aff1Si[0  , 0] := 1.00000E+01; aff1Si[0  , 1] := -9.41486E+00;
aff1Si[1  , 0] := 1.99800E+01; aff1Si[1  , 1] := -1.02392E+01;
aff1Si[2  , 0] := 2.99600E+01; aff1Si[2  , 1] := -1.04800E+01;
aff1Si[3  , 0] := 3.99400E+01; aff1Si[3  , 1] := -1.06753E+01;
aff1Si[4  , 0] := 4.99200E+01; aff1Si[4  , 1] := -1.09200E+01;
aff1Si[5  , 0] := 5.99000E+01; aff1Si[5  , 1] := -1.12738E+01;
aff1Si[6  , 0] := 6.98800E+01; aff1Si[6  , 1] := -1.18088E+01;
aff1Si[7  , 0] := 7.98600E+01; aff1Si[7  , 1] := -1.26670E+01;
aff1Si[8  , 0] := 8.98400E+01; aff1Si[8  , 1] := -1.42966E+01;
aff1Si[9  , 0] := 9.98200E+01; aff1Si[9  , 1] := -2.06210E+01;
aff1Si[10 , 0] := 1.09800E+02; aff1Si[10 , 1] := -1.46441E+01;
aff1Si[11 , 0] := 1.19780E+02; aff1Si[11 , 1] := -1.26978E+01;
aff1Si[12 , 0] := 1.29760E+02; aff1Si[12 , 1] := -1.11702E+01;
aff1Si[13 , 0] := 1.39740E+02; aff1Si[13 , 1] := -9.97819E+00;
aff1Si[14 , 0] := 1.49720E+02; aff1Si[14 , 1] := -9.38400E+00;
aff1Si[15 , 0] := 1.59700E+02; aff1Si[15 , 1] := -7.66375E+00;
aff1Si[16 , 0] := 1.69680E+02; aff1Si[16 , 1] := -6.56070E+00;
aff1Si[17 , 0] := 1.79660E+02; aff1Si[17 , 1] := -5.66709E+00;
aff1Si[18 , 0] := 1.89640E+02; aff1Si[18 , 1] := -4.92348E+00;
aff1Si[19 , 0] := 1.99620E+02; aff1Si[19 , 1] := -4.29899E+00;
aff1Si[20 , 0] := 2.09600E+02; aff1Si[20 , 1] := -3.77192E+00;
aff1Si[21 , 0] := 2.19580E+02; aff1Si[21 , 1] := -3.32553E+00;
aff1Si[22 , 0] := 2.29560E+02; aff1Si[22 , 1] := -2.94654E+00;
aff1Si[23 , 0] := 2.39540E+02; aff1Si[23 , 1] := -2.62393E+00;
aff1Si[24 , 0] := 2.49520E+02; aff1Si[24 , 1] := -2.34859E+00;
aff1Si[25 , 0] := 2.59500E+02; aff1Si[25 , 1] := -2.11303E+00;
aff1Si[26 , 0] := 2.69480E+02; aff1Si[26 , 1] := -1.91106E+00;
aff1Si[27 , 0] := 2.79460E+02; aff1Si[27 , 1] := -1.73755E+00;
aff1Si[28 , 0] := 2.89440E+02; aff1Si[28 , 1] := -1.58823E+00;
aff1Si[29 , 0] := 2.99420E+02; aff1Si[29 , 1] := -1.45933E+00;
aff1Si[30 , 0] := 3.09400E+02; aff1Si[30 , 1] := -1.34828E+00;
aff1Si[31 , 0] := 3.19380E+02; aff1Si[31 , 1] := -1.25237E+00;
aff1Si[32 , 0] := 3.29360E+02; aff1Si[32 , 1] := -1.16949E+00;
aff1Si[33 , 0] := 3.39340E+02; aff1Si[33 , 1] := -1.09787E+00;
aff1Si[34 , 0] := 3.49320E+02; aff1Si[34 , 1] := -1.03599E+00;
aff1Si[35 , 0] := 3.59300E+02; aff1Si[35 , 1] := -9.82554E-01;
aff1Si[36 , 0] := 3.69280E+02; aff1Si[36 , 1] := -9.36462E-01;
aff1Si[37 , 0] := 3.79260E+02; aff1Si[37 , 1] := -8.96770E-01;
aff1Si[38 , 0] := 3.89240E+02; aff1Si[38 , 1] := -8.62629E-01;
aff1Si[39 , 0] := 3.99220E+02; aff1Si[39 , 1] := -8.33381E-01;
aff1Si[40 , 0] := 4.09200E+02; aff1Si[40 , 1] := -8.08424E-01;
aff1Si[41 , 0] := 4.19180E+02; aff1Si[41 , 1] := -7.87310E-01;
aff1Si[42 , 0] := 4.29160E+02; aff1Si[42 , 1] := -7.69634E-01;
aff1Si[43 , 0] := 4.39140E+02; aff1Si[43 , 1] := -7.55027E-01;
aff1Si[44 , 0] := 4.49120E+02; aff1Si[44 , 1] := -7.43244E-01;
aff1Si[45 , 0] := 4.59100E+02; aff1Si[45 , 1] := -7.33827E-01;
aff1Si[46 , 0] := 4.69080E+02; aff1Si[46 , 1] := -7.26554E-01;
aff1Si[47 , 0] := 4.79060E+02; aff1Si[47 , 1] := -7.21214E-01;
aff1Si[48 , 0] := 4.89040E+02; aff1Si[48 , 1] := -7.17596E-01;
aff1Si[49 , 0] := 4.99020E+02; aff1Si[49 , 1] := -7.15514E-01;
aff1Si[50 , 0] := 5.09000E+02; aff1Si[50 , 1] := -7.14800E-01;
aff1Si[51 , 0] := 5.18980E+02; aff1Si[51 , 1] := -7.15307E-01;
aff1Si[52 , 0] := 5.28960E+02; aff1Si[52 , 1] := -7.16904E-01;
aff1Si[53 , 0] := 5.38940E+02; aff1Si[53 , 1] := -7.19472E-01;
aff1Si[54 , 0] := 5.48920E+02; aff1Si[54 , 1] := -7.22908E-01;
aff1Si[55 , 0] := 5.58900E+02; aff1Si[55 , 1] := -7.27117E-01;
aff1Si[56 , 0] := 5.68880E+02; aff1Si[56 , 1] := -7.32017E-01;
aff1Si[57 , 0] := 5.78860E+02; aff1Si[57 , 1] := -7.37532E-01;
aff1Si[58 , 0] := 5.88840E+02; aff1Si[58 , 1] := -7.43594E-01;
aff1Si[59 , 0] := 5.98820E+02; aff1Si[59 , 1] := -7.50144E-01;
aff1Si[60 , 0] := 6.08800E+02; aff1Si[60 , 1] := -7.57132E-01;
aff1Si[61 , 0] := 6.18780E+02; aff1Si[61 , 1] := -7.64516E-01;
aff1Si[62 , 0] := 6.28760E+02; aff1Si[62 , 1] := -7.72258E-01;
aff1Si[63 , 0] := 6.38740E+02; aff1Si[63 , 1] := -7.80324E-01;
aff1Si[64 , 0] := 6.48720E+02; aff1Si[64 , 1] := -7.88682E-01;
aff1Si[65 , 0] := 6.58700E+02; aff1Si[65 , 1] := -7.97301E-01;
aff1Si[66 , 0] := 6.68680E+02; aff1Si[66 , 1] := -8.06156E-01;
aff1Si[67 , 0] := 6.78660E+02; aff1Si[67 , 1] := -8.15222E-01;
aff1Si[68 , 0] := 6.88640E+02; aff1Si[68 , 1] := -8.24477E-01;
aff1Si[69 , 0] := 6.98620E+02; aff1Si[69 , 1] := -8.33900E-01;
aff1Si[70 , 0] := 7.08600E+02; aff1Si[70 , 1] := -8.43475E-01;
aff1Si[71 , 0] := 7.18580E+02; aff1Si[71 , 1] := -8.53184E-01;
aff1Si[72 , 0] := 7.28560E+02; aff1Si[72 , 1] := -8.63013E-01;
aff1Si[73 , 0] := 7.38540E+02; aff1Si[73 , 1] := -8.72949E-01;
aff1Si[74 , 0] := 7.48520E+02; aff1Si[74 , 1] := -8.82980E-01;
aff1Si[75 , 0] := 7.58500E+02; aff1Si[75 , 1] := -8.93095E-01;
aff1Si[76 , 0] := 7.68480E+02; aff1Si[76 , 1] := -9.03283E-01;
aff1Si[77 , 0] := 7.78460E+02; aff1Si[77 , 1] := -9.13538E-01;
aff1Si[78 , 0] := 7.88440E+02; aff1Si[78 , 1] := -9.23850E-01;
aff1Si[79 , 0] := 7.98420E+02; aff1Si[79 , 1] := -9.34213E-01;
aff1Si[80 , 0] := 8.08400E+02; aff1Si[80 , 1] := -9.44619E-01;
aff1Si[81 , 0] := 8.18380E+02; aff1Si[81 , 1] := -9.55065E-01;
aff1Si[82 , 0] := 8.28360E+02; aff1Si[82 , 1] := -9.65543E-01;
aff1Si[83 , 0] := 8.38340E+02; aff1Si[83 , 1] := -9.76051E-01;
aff1Si[84 , 0] := 8.48320E+02; aff1Si[84 , 1] := -9.86582E-01;
aff1Si[85 , 0] := 8.58300E+02; aff1Si[85 , 1] := -9.97133E-01;
aff1Si[86 , 0] := 8.68280E+02; aff1Si[86 , 1] := -1.00770E+00;
aff1Si[87 , 0] := 8.78260E+02; aff1Si[87 , 1] := -1.01828E+00;
aff1Si[88 , 0] := 8.88240E+02; aff1Si[88 , 1] := -1.02887E+00;
aff1Si[89 , 0] := 8.98220E+02; aff1Si[89 , 1] := -1.03946E+00;
aff1Si[90 , 0] := 9.08200E+02; aff1Si[90 , 1] := -1.05006E+00;
aff1Si[91 , 0] := 9.18180E+02; aff1Si[91 , 1] := -1.06065E+00;
aff1Si[92 , 0] := 9.28160E+02; aff1Si[92 , 1] := -1.07124E+00;
aff1Si[93 , 0] := 9.38140E+02; aff1Si[93 , 1] := -1.08181E+00;
aff1Si[94 , 0] := 9.48120E+02; aff1Si[94 , 1] := -1.09236E+00;
aff1Si[95 , 0] := 9.58100E+02; aff1Si[95 , 1] := -1.10289E+00;
aff1Si[96 , 0] := 9.68080E+02; aff1Si[96 , 1] := -1.11339E+00;
aff1Si[97 , 0] := 9.78060E+02; aff1Si[97 , 1] := -1.12383E+00;
aff1Si[98 , 0] := 9.88040E+02; aff1Si[98 , 1] := -1.13422E+00;
aff1Si[99 , 0] := 9.98020E+02; aff1Si[99 , 1] := -1.14454E+00;
aff1Si[100, 0] := 1.00800E+03; aff1Si[100, 1] := -1.15552E+00;
aff1Si[101, 0] := 1.01798E+03; aff1Si[101, 1] := -1.16689E+00;
aff1Si[102, 0] := 1.02796E+03; aff1Si[102, 1] := -1.17846E+00;
aff1Si[103, 0] := 1.03794E+03; aff1Si[103, 1] := -1.19023E+00;
aff1Si[104, 0] := 1.04792E+03; aff1Si[104, 1] := -1.20217E+00;
aff1Si[105, 0] := 1.05790E+03; aff1Si[105, 1] := -1.21429E+00;
aff1Si[106, 0] := 1.06788E+03; aff1Si[106, 1] := -1.22657E+00;
aff1Si[107, 0] := 1.07786E+03; aff1Si[107, 1] := -1.23901E+00;
aff1Si[108, 0] := 1.08784E+03; aff1Si[108, 1] := -1.25161E+00;
aff1Si[109, 0] := 1.09782E+03; aff1Si[109, 1] := -1.26436E+00;
aff1Si[110, 0] := 1.10780E+03; aff1Si[110, 1] := -1.27726E+00;
aff1Si[111, 0] := 1.11778E+03; aff1Si[111, 1] := -1.29031E+00;
aff1Si[112, 0] := 1.12776E+03; aff1Si[112, 1] := -1.30352E+00;
aff1Si[113, 0] := 1.13774E+03; aff1Si[113, 1] := -1.31687E+00;
aff1Si[114, 0] := 1.14772E+03; aff1Si[114, 1] := -1.33039E+00;
aff1Si[115, 0] := 1.15770E+03; aff1Si[115, 1] := -1.34406E+00;
aff1Si[116, 0] := 1.16768E+03; aff1Si[116, 1] := -1.35790E+00;
aff1Si[117, 0] := 1.17766E+03; aff1Si[117, 1] := -1.37190E+00;
aff1Si[118, 0] := 1.18764E+03; aff1Si[118, 1] := -1.38607E+00;
aff1Si[119, 0] := 1.19762E+03; aff1Si[119, 1] := -1.40042E+00;
aff1Si[120, 0] := 1.20760E+03; aff1Si[120, 1] := -1.41495E+00;
aff1Si[121, 0] := 1.21758E+03; aff1Si[121, 1] := -1.42967E+00;
aff1Si[122, 0] := 1.22756E+03; aff1Si[122, 1] := -1.44459E+00;
aff1Si[123, 0] := 1.23754E+03; aff1Si[123, 1] := -1.45971E+00;
aff1Si[124, 0] := 1.24752E+03; aff1Si[124, 1] := -1.47505E+00;
aff1Si[125, 0] := 1.25750E+03; aff1Si[125, 1] := -1.49061E+00;
aff1Si[126, 0] := 1.26748E+03; aff1Si[126, 1] := -1.50640E+00;
aff1Si[127, 0] := 1.27746E+03; aff1Si[127, 1] := -1.52244E+00;
aff1Si[128, 0] := 1.28744E+03; aff1Si[128, 1] := -1.53873E+00;
aff1Si[129, 0] := 1.29742E+03; aff1Si[129, 1] := -1.55528E+00;
aff1Si[130, 0] := 1.30740E+03; aff1Si[130, 1] := -1.57211E+00;
aff1Si[131, 0] := 1.31738E+03; aff1Si[131, 1] := -1.58924E+00;
aff1Si[132, 0] := 1.32736E+03; aff1Si[132, 1] := -1.60667E+00;
aff1Si[133, 0] := 1.33734E+03; aff1Si[133, 1] := -1.62443E+00;
aff1Si[134, 0] := 1.34732E+03; aff1Si[134, 1] := -1.64252E+00;
aff1Si[135, 0] := 1.35730E+03; aff1Si[135, 1] := -1.66096E+00;
aff1Si[136, 0] := 1.36728E+03; aff1Si[136, 1] := -1.67978E+00;
aff1Si[137, 0] := 1.37726E+03; aff1Si[137, 1] := -1.69900E+00;
aff1Si[138, 0] := 1.38724E+03; aff1Si[138, 1] := -1.71863E+00;
aff1Si[139, 0] := 1.39722E+03; aff1Si[139, 1] := -1.73869E+00;
aff1Si[140, 0] := 1.40720E+03; aff1Si[140, 1] := -1.75922E+00;
aff1Si[141, 0] := 1.41718E+03; aff1Si[141, 1] := -1.78024E+00;
aff1Si[142, 0] := 1.42716E+03; aff1Si[142, 1] := -1.80177E+00;
aff1Si[143, 0] := 1.43714E+03; aff1Si[143, 1] := -1.82385E+00;
aff1Si[144, 0] := 1.44712E+03; aff1Si[144, 1] := -1.84650E+00;
aff1Si[145, 0] := 1.45710E+03; aff1Si[145, 1] := -1.86977E+00;
aff1Si[146, 0] := 1.46708E+03; aff1Si[146, 1] := -1.89369E+00;
aff1Si[147, 0] := 1.47706E+03; aff1Si[147, 1] := -1.91830E+00;
aff1Si[148, 0] := 1.48704E+03; aff1Si[148, 1] := -1.94364E+00;
aff1Si[149, 0] := 1.49702E+03; aff1Si[149, 1] := -1.96977E+00;
aff1Si[150, 0] := 1.50700E+03; aff1Si[150, 1] := -1.99674E+00;
aff1Si[151, 0] := 1.51698E+03; aff1Si[151, 1] := -2.02460E+00;
aff1Si[152, 0] := 1.52696E+03; aff1Si[152, 1] := -2.05341E+00;
aff1Si[153, 0] := 1.53694E+03; aff1Si[153, 1] := -2.08326E+00;
aff1Si[154, 0] := 1.54692E+03; aff1Si[154, 1] := -2.11421E+00;
aff1Si[155, 0] := 1.55690E+03; aff1Si[155, 1] := -2.14634E+00;
aff1Si[156, 0] := 1.56688E+03; aff1Si[156, 1] := -2.17976E+00;
aff1Si[157, 0] := 1.57686E+03; aff1Si[157, 1] := -2.21456E+00;
aff1Si[158, 0] := 1.58684E+03; aff1Si[158, 1] := -2.25087E+00;
aff1Si[159, 0] := 1.59682E+03; aff1Si[159, 1] := -2.28882E+00;
aff1Si[160, 0] := 1.60680E+03; aff1Si[160, 1] := -2.32855E+00;
aff1Si[161, 0] := 1.61678E+03; aff1Si[161, 1] := -2.37023E+00;
aff1Si[162, 0] := 1.62676E+03; aff1Si[162, 1] := -2.41406E+00;
aff1Si[163, 0] := 1.63674E+03; aff1Si[163, 1] := -2.46026E+00;
aff1Si[164, 0] := 1.64672E+03; aff1Si[164, 1] := -2.50908E+00;
aff1Si[165, 0] := 1.65670E+03; aff1Si[165, 1] := -2.56082E+00;
aff1Si[166, 0] := 1.66668E+03; aff1Si[166, 1] := -2.61583E+00;
aff1Si[167, 0] := 1.67666E+03; aff1Si[167, 1] := -2.67452E+00;
aff1Si[168, 0] := 1.68664E+03; aff1Si[168, 1] := -2.73738E+00;
aff1Si[169, 0] := 1.69662E+03; aff1Si[169, 1] := -2.80500E+00;
aff1Si[170, 0] := 1.70660E+03; aff1Si[170, 1] := -2.87810E+00;
aff1Si[171, 0] := 1.71658E+03; aff1Si[171, 1] := -2.95759E+00;
aff1Si[172, 0] := 1.72656E+03; aff1Si[172, 1] := -3.04459E+00;
aff1Si[173, 0] := 1.73654E+03; aff1Si[173, 1] := -3.14056E+00;
aff1Si[174, 0] := 1.74652E+03; aff1Si[174, 1] := -3.24738E+00;
aff1Si[175, 0] := 1.75650E+03; aff1Si[175, 1] := -3.36764E+00;
aff1Si[176, 0] := 1.76648E+03; aff1Si[176, 1] := -3.50505E+00;
aff1Si[177, 0] := 1.77646E+03; aff1Si[177, 1] := -3.66418E+00;
aff1Si[178, 0] := 1.78644E+03; aff1Si[178, 1] := -3.85516E+00;
aff1Si[179, 0] := 1.79642E+03; aff1Si[179, 1] := -4.08637E+00;
aff1Si[180, 0] := 1.80640E+03; aff1Si[180, 1] := -4.38853E+00;
aff1Si[181, 0] := 1.81638E+03; aff1Si[181, 1] := -4.79985E+00;
aff1Si[182, 0] := 1.82636E+03; aff1Si[182, 1] := -5.47277E+00;
aff1Si[183, 0] := 1.83634E+03; aff1Si[183, 1] := -7.34626E+00;
aff1Si[184, 0] := 1.84632E+03; aff1Si[184, 1] := -6.10004E+00;
aff1Si[185, 0] := 1.85630E+03; aff1Si[185, 1] := -5.04971E+00;
aff1Si[186, 0] := 1.86628E+03; aff1Si[186, 1] := -4.48521E+00;
aff1Si[187, 0] := 1.87626E+03; aff1Si[187, 1] := -4.09245E+00;
aff1Si[188, 0] := 1.88624E+03; aff1Si[188, 1] := -3.78618E+00;
aff1Si[189, 0] := 1.89622E+03; aff1Si[189, 1] := -3.53446E+00;
aff1Si[190, 0] := 1.90620E+03; aff1Si[190, 1] := -3.32140E+00;
aff1Si[191, 0] := 1.91618E+03; aff1Si[191, 1] := -3.13320E+00;
aff1Si[192, 0] := 1.92616E+03; aff1Si[192, 1] := -2.96477E+00;
aff1Si[193, 0] := 1.93614E+03; aff1Si[193, 1] := -2.81052E+00;
aff1Si[194, 0] := 1.94612E+03; aff1Si[194, 1] := -2.67041E+00;
aff1Si[195, 0] := 1.95610E+03; aff1Si[195, 1] := -2.54343E+00;
aff1Si[196, 0] := 1.96608E+03; aff1Si[196, 1] := -2.42698E+00;
aff1Si[197, 0] := 1.97606E+03; aff1Si[197, 1] := -2.31896E+00;
aff1Si[198, 0] := 1.98604E+03; aff1Si[198, 1] := -2.21841E+00;
aff1Si[199, 0] := 1.99602E+03; aff1Si[199, 1] := -2.12444E+00;
aff1Si[200, 0] := 2.00600E+03; aff1Si[200, 1] := -2.03625E+00;
aff1Si[201, 0] := 2.01598E+03; aff1Si[201, 1] := -1.95322E+00;
aff1Si[202, 0] := 2.02596E+03; aff1Si[202, 1] := -1.87485E+00;
aff1Si[203, 0] := 2.03594E+03; aff1Si[203, 1] := -1.80069E+00;
aff1Si[204, 0] := 2.04592E+03; aff1Si[204, 1] := -1.73037E+00;
aff1Si[205, 0] := 2.05590E+03; aff1Si[205, 1] := -1.66356E+00;
aff1Si[206, 0] := 2.06588E+03; aff1Si[206, 1] := -1.59999E+00;
aff1Si[207, 0] := 2.07586E+03; aff1Si[207, 1] := -1.53941E+00;
aff1Si[208, 0] := 2.08584E+03; aff1Si[208, 1] := -1.48161E+00;
aff1Si[209, 0] := 2.09582E+03; aff1Si[209, 1] := -1.42639E+00;
aff1Si[210, 0] := 2.10580E+03; aff1Si[210, 1] := -1.37358E+00;
aff1Si[211, 0] := 2.11578E+03; aff1Si[211, 1] := -1.32303E+00;
aff1Si[212, 0] := 2.12576E+03; aff1Si[212, 1] := -1.27460E+00;
aff1Si[213, 0] := 2.13574E+03; aff1Si[213, 1] := -1.22815E+00;
aff1Si[214, 0] := 2.14572E+03; aff1Si[214, 1] := -1.18358E+00;
aff1Si[215, 0] := 2.15570E+03; aff1Si[215, 1] := -1.14078E+00;
aff1Si[216, 0] := 2.16568E+03; aff1Si[216, 1] := -1.09965E+00;
aff1Si[217, 0] := 2.17566E+03; aff1Si[217, 1] := -1.06011E+00;
aff1Si[218, 0] := 2.18564E+03; aff1Si[218, 1] := -1.02206E+00;
aff1Si[219, 0] := 2.19562E+03; aff1Si[219, 1] := -9.85443E-01;
aff1Si[220, 0] := 2.20560E+03; aff1Si[220, 1] := -9.50177E-01;
aff1Si[221, 0] := 2.21558E+03; aff1Si[221, 1] := -9.16199E-01;
aff1Si[222, 0] := 2.22556E+03; aff1Si[222, 1] := -8.83447E-01;
aff1Si[223, 0] := 2.23554E+03; aff1Si[223, 1] := -8.51865E-01;
aff1Si[224, 0] := 2.24552E+03; aff1Si[224, 1] := -8.21397E-01;
aff1Si[225, 0] := 2.25550E+03; aff1Si[225, 1] := -7.91995E-01;
aff1Si[226, 0] := 2.26548E+03; aff1Si[226, 1] := -7.63611E-01;
aff1Si[227, 0] := 2.27546E+03; aff1Si[227, 1] := -7.36201E-01;
aff1Si[228, 0] := 2.28544E+03; aff1Si[228, 1] := -7.09723E-01;
aff1Si[229, 0] := 2.29542E+03; aff1Si[229, 1] := -6.84138E-01;
aff1Si[230, 0] := 2.30540E+03; aff1Si[230, 1] := -6.59410E-01;
aff1Si[231, 0] := 2.31538E+03; aff1Si[231, 1] := -6.35505E-01;
aff1Si[232, 0] := 2.32536E+03; aff1Si[232, 1] := -6.12392E-01;
aff1Si[233, 0] := 2.33534E+03; aff1Si[233, 1] := -5.90040E-01;
aff1Si[234, 0] := 2.34532E+03; aff1Si[234, 1] := -5.68423E-01;
aff1Si[235, 0] := 2.35530E+03; aff1Si[235, 1] := -5.47512E-01;
aff1Si[236, 0] := 2.36528E+03; aff1Si[236, 1] := -5.27295E-01;
aff1Si[237, 0] := 2.37526E+03; aff1Si[237, 1] := -5.07776E-01;
aff1Si[238, 0] := 2.38524E+03; aff1Si[238, 1] := -4.88918E-01;
aff1Si[239, 0] := 2.39522E+03; aff1Si[239, 1] := -4.70610E-01;
aff1Si[240, 0] := 2.40520E+03; aff1Si[240, 1] := -4.52760E-01;
aff1Si[241, 0] := 2.41518E+03; aff1Si[241, 1] := -4.35340E-01;
aff1Si[242, 0] := 2.42516E+03; aff1Si[242, 1] := -4.18341E-01;
aff1Si[243, 0] := 2.43514E+03; aff1Si[243, 1] := -4.01751E-01;
aff1Si[244, 0] := 2.44512E+03; aff1Si[244, 1] := -3.85562E-01;
aff1Si[245, 0] := 2.45510E+03; aff1Si[245, 1] := -3.69769E-01;
aff1Si[246, 0] := 2.46508E+03; aff1Si[246, 1] := -3.54360E-01;
aff1Si[247, 0] := 2.47506E+03; aff1Si[247, 1] := -3.39322E-01;
aff1Si[248, 0] := 2.48504E+03; aff1Si[248, 1] := -3.24645E-01;
aff1Si[249, 0] := 2.49502E+03; aff1Si[249, 1] := -3.10317E-01;
aff1Si[250, 0] := 2.50500E+03; aff1Si[250, 1] := -2.96329E-01;
aff1Si[251, 0] := 2.51498E+03; aff1Si[251, 1] := -2.82670E-01;
aff1Si[252, 0] := 2.52496E+03; aff1Si[252, 1] := -2.69329E-01;
aff1Si[253, 0] := 2.53494E+03; aff1Si[253, 1] := -2.56297E-01;
aff1Si[254, 0] := 2.54492E+03; aff1Si[254, 1] := -2.43563E-01;
aff1Si[255, 0] := 2.55490E+03; aff1Si[255, 1] := -2.31120E-01;
aff1Si[256, 0] := 2.56488E+03; aff1Si[256, 1] := -2.18957E-01;
aff1Si[257, 0] := 2.57486E+03; aff1Si[257, 1] := -2.07066E-01;
aff1Si[258, 0] := 2.58484E+03; aff1Si[258, 1] := -1.95440E-01;
aff1Si[259, 0] := 2.59482E+03; aff1Si[259, 1] := -1.84069E-01;
aff1Si[260, 0] := 2.60480E+03; aff1Si[260, 1] := -1.72947E-01;
aff1Si[261, 0] := 2.61478E+03; aff1Si[261, 1] := -1.62065E-01;
aff1Si[262, 0] := 2.62476E+03; aff1Si[262, 1] := -1.51417E-01;
aff1Si[263, 0] := 2.63474E+03; aff1Si[263, 1] := -1.40996E-01;
aff1Si[264, 0] := 2.64472E+03; aff1Si[264, 1] := -1.30795E-01;
aff1Si[265, 0] := 2.65470E+03; aff1Si[265, 1] := -1.20808E-01;
aff1Si[266, 0] := 2.66468E+03; aff1Si[266, 1] := -1.11029E-01;
aff1Si[267, 0] := 2.67466E+03; aff1Si[267, 1] := -1.01451E-01;
aff1Si[268, 0] := 2.68464E+03; aff1Si[268, 1] := -9.20694E-02;
aff1Si[269, 0] := 2.69462E+03; aff1Si[269, 1] := -8.28782E-02;
aff1Si[270, 0] := 2.70460E+03; aff1Si[270, 1] := -7.38721E-02;
aff1Si[271, 0] := 2.71458E+03; aff1Si[271, 1] := -6.50458E-02;
aff1Si[272, 0] := 2.72456E+03; aff1Si[272, 1] := -5.63945E-02;
aff1Si[273, 0] := 2.73454E+03; aff1Si[273, 1] := -4.79132E-02;
aff1Si[274, 0] := 2.74452E+03; aff1Si[274, 1] := -3.95973E-02;
aff1Si[275, 0] := 2.75450E+03; aff1Si[275, 1] := -3.14421E-02;
aff1Si[276, 0] := 2.76448E+03; aff1Si[276, 1] := -2.34435E-02;
aff1Si[277, 0] := 2.77446E+03; aff1Si[277, 1] := -1.55966E-02;
aff1Si[278, 0] := 2.78444E+03; aff1Si[278, 1] := -7.89668E-03;
aff1Si[279, 0] := 2.79442E+03; aff1Si[279, 1] := -3.39740E-04;
aff1Si[280, 0] := 2.80440E+03; aff1Si[280, 1] := 7.07698E-03;
aff1Si[281, 0] := 2.81438E+03; aff1Si[281, 1] := 1.43563E-02;
aff1Si[282, 0] := 2.82436E+03; aff1Si[282, 1] := 2.15016E-02;
aff1Si[283, 0] := 2.83434E+03; aff1Si[283, 1] := 2.85169E-02;
aff1Si[284, 0] := 2.84432E+03; aff1Si[284, 1] := 3.54063E-02;
aff1Si[285, 0] := 2.85430E+03; aff1Si[285, 1] := 4.21738E-02;
aff1Si[286, 0] := 2.86428E+03; aff1Si[286, 1] := 4.88234E-02;
aff1Si[287, 0] := 2.87426E+03; aff1Si[287, 1] := 5.53597E-02;
aff1Si[288, 0] := 2.88424E+03; aff1Si[288, 1] := 6.17870E-02;
aff1Si[289, 0] := 2.89422E+03; aff1Si[289, 1] := 6.81096E-02;
aff1Si[290, 0] := 2.90420E+03; aff1Si[290, 1] := 7.43335E-02;
aff1Si[291, 0] := 2.91418E+03; aff1Si[291, 1] := 8.04634E-02;
aff1Si[292, 0] := 2.92416E+03; aff1Si[292, 1] := 8.65042E-02;
aff1Si[293, 0] := 2.93414E+03; aff1Si[293, 1] := 9.24599E-02;
aff1Si[294, 0] := 2.94412E+03; aff1Si[294, 1] := 9.83497E-02;
aff1Si[295, 0] := 2.95410E+03; aff1Si[295, 1] := 1.04190E-01;
aff1Si[296, 0] := 2.96408E+03; aff1Si[296, 1] := 1.09986E-01;
aff1Si[297, 0] := 2.97406E+03; aff1Si[297, 1] := 1.15743E-01;
aff1Si[298, 0] := 2.98404E+03; aff1Si[298, 1] := 1.21471E-01;
aff1Si[299, 0] := 2.99402E+03; aff1Si[299, 1] := 1.27161E-01;
aff1Si[300, 0] := 3.00400E+03; aff1Si[300, 1] := 1.32716E-01;
aff1Si[301, 0] := 3.01398E+03; aff1Si[301, 1] := 1.38037E-01;
aff1Si[302, 0] := 3.02396E+03; aff1Si[302, 1] := 1.43078E-01;
aff1Si[303, 0] := 3.03394E+03; aff1Si[303, 1] := 1.47916E-01;
aff1Si[304, 0] := 3.04392E+03; aff1Si[304, 1] := 1.52633E-01;
aff1Si[305, 0] := 3.05390E+03; aff1Si[305, 1] := 1.57281E-01;
aff1Si[306, 0] := 3.06388E+03; aff1Si[306, 1] := 1.61844E-01;
aff1Si[307, 0] := 3.07386E+03; aff1Si[307, 1] := 1.66305E-01;
aff1Si[308, 0] := 3.08384E+03; aff1Si[308, 1] := 1.70654E-01;
aff1Si[309, 0] := 3.09382E+03; aff1Si[309, 1] := 1.74903E-01;
aff1Si[310, 0] := 3.10380E+03; aff1Si[310, 1] := 1.79060E-01;
aff1Si[311, 0] := 3.11378E+03; aff1Si[311, 1] := 1.83130E-01;
aff1Si[312, 0] := 3.12376E+03; aff1Si[312, 1] := 1.87113E-01;
aff1Si[313, 0] := 3.13374E+03; aff1Si[313, 1] := 1.91011E-01;
aff1Si[314, 0] := 3.14372E+03; aff1Si[314, 1] := 1.94825E-01;
aff1Si[315, 0] := 3.15370E+03; aff1Si[315, 1] := 1.98557E-01;
aff1Si[316, 0] := 3.16368E+03; aff1Si[316, 1] := 2.02211E-01;
aff1Si[317, 0] := 3.17366E+03; aff1Si[317, 1] := 2.05787E-01;
aff1Si[318, 0] := 3.18364E+03; aff1Si[318, 1] := 2.09289E-01;
aff1Si[319, 0] := 3.19362E+03; aff1Si[319, 1] := 2.12719E-01;
aff1Si[320, 0] := 3.20360E+03; aff1Si[320, 1] := 2.16077E-01;
aff1Si[321, 0] := 3.21358E+03; aff1Si[321, 1] := 2.19365E-01;
aff1Si[322, 0] := 3.22356E+03; aff1Si[322, 1] := 2.22587E-01;
aff1Si[323, 0] := 3.23354E+03; aff1Si[323, 1] := 2.25742E-01;
aff1Si[324, 0] := 3.24352E+03; aff1Si[324, 1] := 2.28833E-01;
aff1Si[325, 0] := 3.25350E+03; aff1Si[325, 1] := 2.31861E-01;
aff1Si[326, 0] := 3.26348E+03; aff1Si[326, 1] := 2.34829E-01;
aff1Si[327, 0] := 3.27346E+03; aff1Si[327, 1] := 2.37736E-01;
aff1Si[328, 0] := 3.28344E+03; aff1Si[328, 1] := 2.40585E-01;
aff1Si[329, 0] := 3.29342E+03; aff1Si[329, 1] := 2.43378E-01;
aff1Si[330, 0] := 3.30340E+03; aff1Si[330, 1] := 2.46114E-01;
aff1Si[331, 0] := 3.31338E+03; aff1Si[331, 1] := 2.48797E-01;
aff1Si[332, 0] := 3.32336E+03; aff1Si[332, 1] := 2.51426E-01;
aff1Si[333, 0] := 3.33334E+03; aff1Si[333, 1] := 2.54004E-01;
aff1Si[334, 0] := 3.34332E+03; aff1Si[334, 1] := 2.56531E-01;
aff1Si[335, 0] := 3.35330E+03; aff1Si[335, 1] := 2.59009E-01;
aff1Si[336, 0] := 3.36328E+03; aff1Si[336, 1] := 2.61439E-01;
aff1Si[337, 0] := 3.37326E+03; aff1Si[337, 1] := 2.63822E-01;
aff1Si[338, 0] := 3.38324E+03; aff1Si[338, 1] := 2.66159E-01;
aff1Si[339, 0] := 3.39322E+03; aff1Si[339, 1] := 2.68451E-01;
aff1Si[340, 0] := 3.40320E+03; aff1Si[340, 1] := 2.70699E-01;
aff1Si[341, 0] := 3.41318E+03; aff1Si[341, 1] := 2.72905E-01;
aff1Si[342, 0] := 3.42316E+03; aff1Si[342, 1] := 2.75069E-01;
aff1Si[343, 0] := 3.43314E+03; aff1Si[343, 1] := 2.77192E-01;
aff1Si[344, 0] := 3.44312E+03; aff1Si[344, 1] := 2.79275E-01;
aff1Si[345, 0] := 3.45310E+03; aff1Si[345, 1] := 2.81320E-01;
aff1Si[346, 0] := 3.46308E+03; aff1Si[346, 1] := 2.83326E-01;
aff1Si[347, 0] := 3.47306E+03; aff1Si[347, 1] := 2.85296E-01;
aff1Si[348, 0] := 3.48304E+03; aff1Si[348, 1] := 2.87230E-01;
aff1Si[349, 0] := 3.49302E+03; aff1Si[349, 1] := 2.89129E-01;
aff1Si[350, 0] := 3.50300E+03; aff1Si[350, 1] := 2.90993E-01;
aff1Si[351, 0] := 3.51298E+03; aff1Si[351, 1] := 2.92824E-01;
aff1Si[352, 0] := 3.52296E+03; aff1Si[352, 1] := 2.94623E-01;
aff1Si[353, 0] := 3.53294E+03; aff1Si[353, 1] := 2.96390E-01;
aff1Si[354, 0] := 3.54292E+03; aff1Si[354, 1] := 2.98126E-01;
aff1Si[355, 0] := 3.55290E+03; aff1Si[355, 1] := 2.99832E-01;
aff1Si[356, 0] := 3.56288E+03; aff1Si[356, 1] := 3.01509E-01;
aff1Si[357, 0] := 3.57286E+03; aff1Si[357, 1] := 3.03158E-01;
aff1Si[358, 0] := 3.58284E+03; aff1Si[358, 1] := 3.04779E-01;
aff1Si[359, 0] := 3.59282E+03; aff1Si[359, 1] := 3.06374E-01;
aff1Si[360, 0] := 3.60280E+03; aff1Si[360, 1] := 3.07977E-01;
aff1Si[361, 0] := 3.61278E+03; aff1Si[361, 1] := 3.09848E-01;
aff1Si[362, 0] := 3.62276E+03; aff1Si[362, 1] := 3.11580E-01;
aff1Si[363, 0] := 3.63274E+03; aff1Si[363, 1] := 3.12856E-01;
aff1Si[364, 0] := 3.64272E+03; aff1Si[364, 1] := 3.12880E-01;
aff1Si[365, 0] := 3.65270E+03; aff1Si[365, 1] := 3.12065E-01;
aff1Si[366, 0] := 3.66268E+03; aff1Si[366, 1] := 3.12868E-01;
aff1Si[367, 0] := 3.67266E+03; aff1Si[367, 1] := 3.17483E-01;
aff1Si[368, 0] := 3.68264E+03; aff1Si[368, 1] := 3.28681E-01;
aff1Si[369, 0] := 3.69262E+03; aff1Si[369, 1] := 3.43861E-01;
aff1Si[370, 0] := 3.70260E+03; aff1Si[370, 1] := 3.59088E-01;
aff1Si[371, 0] := 3.71258E+03; aff1Si[371, 1] := 3.70424E-01;
aff1Si[372, 0] := 3.72256E+03; aff1Si[372, 1] := 3.75142E-01;
aff1Si[373, 0] := 3.73254E+03; aff1Si[373, 1] := 3.75520E-01;
aff1Si[374, 0] := 3.74252E+03; aff1Si[374, 1] := 3.73965E-01;
aff1Si[375, 0] := 3.75250E+03; aff1Si[375, 1] := 3.73012E-01;
aff1Si[376, 0] := 3.76248E+03; aff1Si[376, 1] := 3.73580E-01;
aff1Si[377, 0] := 3.77246E+03; aff1Si[377, 1] := 3.74958E-01;
aff1Si[378, 0] := 3.78244E+03; aff1Si[378, 1] := 3.76594E-01;
aff1Si[379, 0] := 3.79242E+03; aff1Si[379, 1] := 3.77834E-01;
aff1Si[380, 0] := 3.80240E+03; aff1Si[380, 1] := 3.78780E-01;
aff1Si[381, 0] := 3.81238E+03; aff1Si[381, 1] := 3.79589E-01;
aff1Si[382, 0] := 3.82236E+03; aff1Si[382, 1] := 3.80342E-01;
aff1Si[383, 0] := 3.83234E+03; aff1Si[383, 1] := 3.81150E-01;
aff1Si[384, 0] := 3.84232E+03; aff1Si[384, 1] := 3.81934E-01;
aff1Si[385, 0] := 3.85230E+03; aff1Si[385, 1] := 3.82688E-01;
aff1Si[386, 0] := 3.86228E+03; aff1Si[386, 1] := 3.83414E-01;
aff1Si[387, 0] := 3.87226E+03; aff1Si[387, 1] := 3.84112E-01;
aff1Si[388, 0] := 3.88224E+03; aff1Si[388, 1] := 3.84783E-01;
aff1Si[389, 0] := 3.89222E+03; aff1Si[389, 1] := 3.85427E-01;
aff1Si[390, 0] := 3.90220E+03; aff1Si[390, 1] := 3.86046E-01;
aff1Si[391, 0] := 3.91218E+03; aff1Si[391, 1] := 3.86640E-01;
aff1Si[392, 0] := 3.92216E+03; aff1Si[392, 1] := 3.87210E-01;
aff1Si[393, 0] := 3.93214E+03; aff1Si[393, 1] := 3.87756E-01;
aff1Si[394, 0] := 3.94212E+03; aff1Si[394, 1] := 3.88279E-01;
aff1Si[395, 0] := 3.95210E+03; aff1Si[395, 1] := 3.88779E-01;
aff1Si[396, 0] := 3.96208E+03; aff1Si[396, 1] := 3.89258E-01;
aff1Si[397, 0] := 3.97206E+03; aff1Si[397, 1] := 3.89715E-01;
aff1Si[398, 0] := 3.98204E+03; aff1Si[398, 1] := 3.90152E-01;
aff1Si[399, 0] := 3.99202E+03; aff1Si[399, 1] := 3.90568E-01;
aff1Si[400, 0] := 4.00200E+03; aff1Si[400, 1] := 3.90964E-01;
aff1Si[401, 0] := 4.01198E+03; aff1Si[401, 1] := 3.91341E-01;
aff1Si[402, 0] := 4.02196E+03; aff1Si[402, 1] := 3.91699E-01;
aff1Si[403, 0] := 4.03194E+03; aff1Si[403, 1] := 3.92038E-01;
aff1Si[404, 0] := 4.04192E+03; aff1Si[404, 1] := 3.92359E-01;
aff1Si[405, 0] := 4.05190E+03; aff1Si[405, 1] := 3.92663E-01;
aff1Si[406, 0] := 4.06188E+03; aff1Si[406, 1] := 3.92949E-01;
aff1Si[407, 0] := 4.07186E+03; aff1Si[407, 1] := 3.93219E-01;
aff1Si[408, 0] := 4.08184E+03; aff1Si[408, 1] := 3.93472E-01;
aff1Si[409, 0] := 4.09182E+03; aff1Si[409, 1] := 3.93708E-01;
aff1Si[410, 0] := 4.10180E+03; aff1Si[410, 1] := 3.93929E-01;
aff1Si[411, 0] := 4.11178E+03; aff1Si[411, 1] := 3.94135E-01;
aff1Si[412, 0] := 4.12176E+03; aff1Si[412, 1] := 3.94325E-01;
aff1Si[413, 0] := 4.13174E+03; aff1Si[413, 1] := 3.94501E-01;
aff1Si[414, 0] := 4.14172E+03; aff1Si[414, 1] := 3.94662E-01;
aff1Si[415, 0] := 4.15170E+03; aff1Si[415, 1] := 3.94809E-01;
aff1Si[416, 0] := 4.16168E+03; aff1Si[416, 1] := 3.94942E-01;
aff1Si[417, 0] := 4.17166E+03; aff1Si[417, 1] := 3.95062E-01;
aff1Si[418, 0] := 4.18164E+03; aff1Si[418, 1] := 3.95168E-01;
aff1Si[419, 0] := 4.19162E+03; aff1Si[419, 1] := 3.95262E-01;
aff1Si[420, 0] := 4.20160E+03; aff1Si[420, 1] := 3.95342E-01;
aff1Si[421, 0] := 4.21158E+03; aff1Si[421, 1] := 3.95411E-01;
aff1Si[422, 0] := 4.22156E+03; aff1Si[422, 1] := 3.95467E-01;
aff1Si[423, 0] := 4.23154E+03; aff1Si[423, 1] := 3.95511E-01;
aff1Si[424, 0] := 4.24152E+03; aff1Si[424, 1] := 3.95543E-01;
aff1Si[425, 0] := 4.25150E+03; aff1Si[425, 1] := 3.95564E-01;
aff1Si[426, 0] := 4.26148E+03; aff1Si[426, 1] := 3.95574E-01;
aff1Si[427, 0] := 4.27146E+03; aff1Si[427, 1] := 3.95572E-01;
aff1Si[428, 0] := 4.28144E+03; aff1Si[428, 1] := 3.95560E-01;
aff1Si[429, 0] := 4.29142E+03; aff1Si[429, 1] := 3.95538E-01;
aff1Si[430, 0] := 4.30140E+03; aff1Si[430, 1] := 3.95505E-01;
aff1Si[431, 0] := 4.31138E+03; aff1Si[431, 1] := 3.95462E-01;
aff1Si[432, 0] := 4.32136E+03; aff1Si[432, 1] := 3.95409E-01;
aff1Si[433, 0] := 4.33134E+03; aff1Si[433, 1] := 3.95346E-01;
aff1Si[434, 0] := 4.34132E+03; aff1Si[434, 1] := 3.95274E-01;
aff1Si[435, 0] := 4.35130E+03; aff1Si[435, 1] := 3.95193E-01;
aff1Si[436, 0] := 4.36128E+03; aff1Si[436, 1] := 3.95102E-01;
aff1Si[437, 0] := 4.37126E+03; aff1Si[437, 1] := 3.95002E-01;
aff1Si[438, 0] := 4.38124E+03; aff1Si[438, 1] := 3.94894E-01;
aff1Si[439, 0] := 4.39122E+03; aff1Si[439, 1] := 3.94777E-01;
aff1Si[440, 0] := 4.40120E+03; aff1Si[440, 1] := 3.94652E-01;
aff1Si[441, 0] := 4.41118E+03; aff1Si[441, 1] := 3.94518E-01;
aff1Si[442, 0] := 4.42116E+03; aff1Si[442, 1] := 3.94377E-01;
aff1Si[443, 0] := 4.43114E+03; aff1Si[443, 1] := 3.94227E-01;
aff1Si[444, 0] := 4.44112E+03; aff1Si[444, 1] := 3.94070E-01;
aff1Si[445, 0] := 4.45110E+03; aff1Si[445, 1] := 3.93905E-01;
aff1Si[446, 0] := 4.46108E+03; aff1Si[446, 1] := 3.93732E-01;
aff1Si[447, 0] := 4.47106E+03; aff1Si[447, 1] := 3.93553E-01;
aff1Si[448, 0] := 4.48104E+03; aff1Si[448, 1] := 3.93366E-01;
aff1Si[449, 0] := 4.49102E+03; aff1Si[449, 1] := 3.93172E-01;
aff1Si[450, 0] := 4.50100E+03; aff1Si[450, 1] := 3.92971E-01;
aff1Si[451, 0] := 4.51098E+03; aff1Si[451, 1] := 3.92764E-01;
aff1Si[452, 0] := 4.52096E+03; aff1Si[452, 1] := 3.92550E-01;
aff1Si[453, 0] := 4.53094E+03; aff1Si[453, 1] := 3.92330E-01;
aff1Si[454, 0] := 4.54092E+03; aff1Si[454, 1] := 3.92103E-01;
aff1Si[455, 0] := 4.55090E+03; aff1Si[455, 1] := 3.91870E-01;
aff1Si[456, 0] := 4.56088E+03; aff1Si[456, 1] := 3.91631E-01;
aff1Si[457, 0] := 4.57086E+03; aff1Si[457, 1] := 3.91386E-01;
aff1Si[458, 0] := 4.58084E+03; aff1Si[458, 1] := 3.91135E-01;
aff1Si[459, 0] := 4.59082E+03; aff1Si[459, 1] := 3.90878E-01;
aff1Si[460, 0] := 4.60080E+03; aff1Si[460, 1] := 3.90616E-01;
aff1Si[461, 0] := 4.61078E+03; aff1Si[461, 1] := 3.90348E-01;
aff1Si[462, 0] := 4.62076E+03; aff1Si[462, 1] := 3.90075E-01;
aff1Si[463, 0] := 4.63074E+03; aff1Si[463, 1] := 3.89797E-01;
aff1Si[464, 0] := 4.64072E+03; aff1Si[464, 1] := 3.89513E-01;
aff1Si[465, 0] := 4.65070E+03; aff1Si[465, 1] := 3.89225E-01;
aff1Si[466, 0] := 4.66068E+03; aff1Si[466, 1] := 3.88931E-01;
aff1Si[467, 0] := 4.67066E+03; aff1Si[467, 1] := 3.88633E-01;
aff1Si[468, 0] := 4.68064E+03; aff1Si[468, 1] := 3.88330E-01;
aff1Si[469, 0] := 4.69062E+03; aff1Si[469, 1] := 3.88022E-01;
aff1Si[470, 0] := 4.70060E+03; aff1Si[470, 1] := 3.87710E-01;
aff1Si[471, 0] := 4.71058E+03; aff1Si[471, 1] := 3.87393E-01;
aff1Si[472, 0] := 4.72056E+03; aff1Si[472, 1] := 3.87072E-01;
aff1Si[473, 0] := 4.73054E+03; aff1Si[473, 1] := 3.86746E-01;
aff1Si[474, 0] := 4.74052E+03; aff1Si[474, 1] := 3.86417E-01;
aff1Si[475, 0] := 4.75050E+03; aff1Si[475, 1] := 3.86083E-01;
aff1Si[476, 0] := 4.76048E+03; aff1Si[476, 1] := 3.85745E-01;
aff1Si[477, 0] := 4.77046E+03; aff1Si[477, 1] := 3.85404E-01;
aff1Si[478, 0] := 4.78044E+03; aff1Si[478, 1] := 3.85058E-01;
aff1Si[479, 0] := 4.79042E+03; aff1Si[479, 1] := 3.84709E-01;
aff1Si[480, 0] := 4.80040E+03; aff1Si[480, 1] := 3.84356E-01;
aff1Si[481, 0] := 4.81038E+03; aff1Si[481, 1] := 3.83999E-01;
aff1Si[482, 0] := 4.82036E+03; aff1Si[482, 1] := 3.83639E-01;
aff1Si[483, 0] := 4.83034E+03; aff1Si[483, 1] := 3.83276E-01;
aff1Si[484, 0] := 4.84032E+03; aff1Si[484, 1] := 3.82909E-01;
aff1Si[485, 0] := 4.85030E+03; aff1Si[485, 1] := 3.82538E-01;
aff1Si[486, 0] := 4.86028E+03; aff1Si[486, 1] := 3.82165E-01;
aff1Si[487, 0] := 4.87026E+03; aff1Si[487, 1] := 3.81788E-01;
aff1Si[488, 0] := 4.88024E+03; aff1Si[488, 1] := 3.81409E-01;
aff1Si[489, 0] := 4.89022E+03; aff1Si[489, 1] := 3.81026E-01;
aff1Si[490, 0] := 4.90020E+03; aff1Si[490, 1] := 3.80640E-01;
aff1Si[491, 0] := 4.91018E+03; aff1Si[491, 1] := 3.80251E-01;
aff1Si[492, 0] := 4.92016E+03; aff1Si[492, 1] := 3.79860E-01;
aff1Si[493, 0] := 4.93014E+03; aff1Si[493, 1] := 3.79466E-01;
aff1Si[494, 0] := 4.94012E+03; aff1Si[494, 1] := 3.79069E-01;
aff1Si[495, 0] := 4.95010E+03; aff1Si[495, 1] := 3.78669E-01;
aff1Si[496, 0] := 4.96008E+03; aff1Si[496, 1] := 3.78267E-01;
aff1Si[497, 0] := 4.97006E+03; aff1Si[497, 1] := 3.77862E-01;
aff1Si[498, 0] := 4.98004E+03; aff1Si[498, 1] := 3.77455E-01;
aff1Si[499, 0] := 4.99002E+03; aff1Si[499, 1] := 3.77045E-01;
aff1Si[500, 0] := 5.00000E+03; aff1Si[500, 1] := 3.76633E-01;
aff1Si[501, 0] := 5.05000E+03; aff1Si[501, 1] := 3.74536E-01;
aff1Si[502, 0] := 5.10000E+03; aff1Si[502, 1] := 3.72381E-01;
aff1Si[503, 0] := 5.15000E+03; aff1Si[503, 1] := 3.70187E-01;
aff1Si[504, 0] := 5.20000E+03; aff1Si[504, 1] := 3.67954E-01;
aff1Si[505, 0] := 5.25000E+03; aff1Si[505, 1] := 3.65686E-01;
aff1Si[506, 0] := 5.30000E+03; aff1Si[506, 1] := 3.63389E-01;
aff1Si[507, 0] := 5.35000E+03; aff1Si[507, 1] := 3.61065E-01;
aff1Si[508, 0] := 5.40000E+03; aff1Si[508, 1] := 3.58720E-01;
aff1Si[509, 0] := 5.45000E+03; aff1Si[509, 1] := 3.56357E-01;
aff1Si[510, 0] := 5.50000E+03; aff1Si[510, 1] := 3.53979E-01;
aff1Si[511, 0] := 5.55000E+03; aff1Si[511, 1] := 3.51590E-01;
aff1Si[512, 0] := 5.60000E+03; aff1Si[512, 1] := 3.49191E-01;
aff1Si[513, 0] := 5.65000E+03; aff1Si[513, 1] := 3.46787E-01;
aff1Si[514, 0] := 5.70000E+03; aff1Si[514, 1] := 3.44378E-01;
aff1Si[515, 0] := 5.75000E+03; aff1Si[515, 1] := 3.41968E-01;
aff1Si[516, 0] := 5.80000E+03; aff1Si[516, 1] := 3.39559E-01;
aff1Si[517, 0] := 5.85000E+03; aff1Si[517, 1] := 3.37151E-01;
aff1Si[518, 0] := 5.90000E+03; aff1Si[518, 1] := 3.34748E-01;
aff1Si[519, 0] := 5.95000E+03; aff1Si[519, 1] := 3.32351E-01;
aff1Si[520, 0] := 6.00000E+03; aff1Si[520, 1] := 3.29960E-01;
aff1Si[521, 0] := 6.05000E+03; aff1Si[521, 1] := 3.27578E-01;
aff1Si[522, 0] := 6.10000E+03; aff1Si[522, 1] := 3.25206E-01;
aff1Si[523, 0] := 6.15000E+03; aff1Si[523, 1] := 3.22844E-01;
aff1Si[524, 0] := 6.20000E+03; aff1Si[524, 1] := 3.20494E-01;
aff1Si[525, 0] := 6.25000E+03; aff1Si[525, 1] := 3.18157E-01;
aff1Si[526, 0] := 6.30000E+03; aff1Si[526, 1] := 3.15834E-01;
aff1Si[527, 0] := 6.35000E+03; aff1Si[527, 1] := 3.13524E-01;
aff1Si[528, 0] := 6.40000E+03; aff1Si[528, 1] := 3.11230E-01;
aff1Si[529, 0] := 6.45000E+03; aff1Si[529, 1] := 3.08952E-01;
aff1Si[530, 0] := 6.50000E+03; aff1Si[530, 1] := 3.06691E-01;
aff1Si[531, 0] := 6.55000E+03; aff1Si[531, 1] := 3.04446E-01;
aff1Si[532, 0] := 6.60000E+03; aff1Si[532, 1] := 3.02219E-01;
aff1Si[533, 0] := 6.65000E+03; aff1Si[533, 1] := 3.00010E-01;
aff1Si[534, 0] := 6.70000E+03; aff1Si[534, 1] := 2.97819E-01;
aff1Si[535, 0] := 6.75000E+03; aff1Si[535, 1] := 2.95647E-01;
aff1Si[536, 0] := 6.80000E+03; aff1Si[536, 1] := 2.93494E-01;
aff1Si[537, 0] := 6.85000E+03; aff1Si[537, 1] := 2.91361E-01;
aff1Si[538, 0] := 6.90000E+03; aff1Si[538, 1] := 2.89248E-01;
aff1Si[539, 0] := 6.95000E+03; aff1Si[539, 1] := 2.87154E-01;
aff1Si[540, 0] := 7.00000E+03; aff1Si[540, 1] := 2.85082E-01;
aff1Si[541, 0] := 7.05000E+03; aff1Si[541, 1] := 2.83029E-01;
aff1Si[542, 0] := 7.10000E+03; aff1Si[542, 1] := 2.80998E-01;
aff1Si[543, 0] := 7.15000E+03; aff1Si[543, 1] := 2.78988E-01;
aff1Si[544, 0] := 7.20000E+03; aff1Si[544, 1] := 2.76999E-01;
aff1Si[545, 0] := 7.25000E+03; aff1Si[545, 1] := 2.75032E-01;
aff1Si[546, 0] := 7.30000E+03; aff1Si[546, 1] := 2.73086E-01;
aff1Si[547, 0] := 7.35000E+03; aff1Si[547, 1] := 2.71163E-01;
aff1Si[548, 0] := 7.40000E+03; aff1Si[548, 1] := 2.69262E-01;
aff1Si[549, 0] := 7.45000E+03; aff1Si[549, 1] := 2.67383E-01;
aff1Si[550, 0] := 7.50000E+03; aff1Si[550, 1] := 2.65526E-01;
aff1Si[551, 0] := 7.55000E+03; aff1Si[551, 1] := 2.63693E-01;
aff1Si[552, 0] := 7.60000E+03; aff1Si[552, 1] := 2.61883E-01;
aff1Si[553, 0] := 7.65000E+03; aff1Si[553, 1] := 2.60096E-01;
aff1Si[554, 0] := 7.70000E+03; aff1Si[554, 1] := 2.58333E-01;
aff1Si[555, 0] := 7.75000E+03; aff1Si[555, 1] := 2.56594E-01;
aff1Si[556, 0] := 7.80000E+03; aff1Si[556, 1] := 2.54879E-01;
aff1Si[557, 0] := 7.85000E+03; aff1Si[557, 1] := 2.53189E-01;
aff1Si[558, 0] := 7.90000E+03; aff1Si[558, 1] := 2.51525E-01;
aff1Si[559, 0] := 7.95000E+03; aff1Si[559, 1] := 2.49888E-01;
aff1Si[560, 0] := 8.00000E+03; aff1Si[560, 1] := 2.48273E-01;
aff1Si[561, 0] := 8.05000E+03; aff1Si[561, 1] := 2.46671E-01;
aff1Si[562, 0] := 8.10000E+03; aff1Si[562, 1] := 2.45076E-01;
aff1Si[563, 0] := 8.15000E+03; aff1Si[563, 1] := 2.43488E-01;
aff1Si[564, 0] := 8.20000E+03; aff1Si[564, 1] := 2.41911E-01;
aff1Si[565, 0] := 8.25000E+03; aff1Si[565, 1] := 2.40345E-01;
aff1Si[566, 0] := 8.30000E+03; aff1Si[566, 1] := 2.38792E-01;
aff1Si[567, 0] := 8.35000E+03; aff1Si[567, 1] := 2.37253E-01;
aff1Si[568, 0] := 8.40000E+03; aff1Si[568, 1] := 2.35730E-01;
aff1Si[569, 0] := 8.45000E+03; aff1Si[569, 1] := 2.34224E-01;
aff1Si[570, 0] := 8.50000E+03; aff1Si[570, 1] := 2.32736E-01;
aff1Si[571, 0] := 8.55000E+03; aff1Si[571, 1] := 2.31268E-01;
aff1Si[572, 0] := 8.60000E+03; aff1Si[572, 1] := 2.29822E-01;
aff1Si[573, 0] := 8.65000E+03; aff1Si[573, 1] := 2.28400E-01;
aff1Si[574, 0] := 8.70000E+03; aff1Si[574, 1] := 2.27003E-01;
aff1Si[575, 0] := 8.75000E+03; aff1Si[575, 1] := 2.25634E-01;
aff1Si[576, 0] := 8.80000E+03; aff1Si[576, 1] := 2.24296E-01;
aff1Si[577, 0] := 8.85000E+03; aff1Si[577, 1] := 2.23015E-01;
aff1Si[578, 0] := 8.90000E+03; aff1Si[578, 1] := 2.21719E-01;
aff1Si[579, 0] := 8.95000E+03; aff1Si[579, 1] := 2.20268E-01;
aff1Si[580, 0] := 9.00000E+03; aff1Si[580, 1] := 2.18736E-01;
aff1Si[581, 0] := 9.05000E+03; aff1Si[581, 1] := 2.17241E-01;
aff1Si[582, 0] := 9.10000E+03; aff1Si[582, 1] := 2.15766E-01;
aff1Si[583, 0] := 9.15000E+03; aff1Si[583, 1] := 2.14291E-01;
aff1Si[584, 0] := 9.20000E+03; aff1Si[584, 1] := 2.12822E-01;
aff1Si[585, 0] := 9.25000E+03; aff1Si[585, 1] := 2.11363E-01;
aff1Si[586, 0] := 9.30000E+03; aff1Si[586, 1] := 2.09912E-01;
aff1Si[587, 0] := 9.35000E+03; aff1Si[587, 1] := 2.08470E-01;
aff1Si[588, 0] := 9.40000E+03; aff1Si[588, 1] := 2.07037E-01;
aff1Si[589, 0] := 9.45000E+03; aff1Si[589, 1] := 2.05613E-01;
aff1Si[590, 0] := 9.50000E+03; aff1Si[590, 1] := 2.04198E-01;
aff1Si[591, 0] := 9.55000E+03; aff1Si[591, 1] := 2.02793E-01;
aff1Si[592, 0] := 9.60000E+03; aff1Si[592, 1] := 2.01397E-01;
aff1Si[593, 0] := 9.65000E+03; aff1Si[593, 1] := 2.00010E-01;
aff1Si[594, 0] := 9.70000E+03; aff1Si[594, 1] := 1.98634E-01;
aff1Si[595, 0] := 9.75000E+03; aff1Si[595, 1] := 1.97267E-01;
aff1Si[596, 0] := 9.80000E+03; aff1Si[596, 1] := 1.95910E-01;
aff1Si[597, 0] := 9.85000E+03; aff1Si[597, 1] := 1.94563E-01;
aff1Si[598, 0] := 9.90000E+03; aff1Si[598, 1] := 1.93226E-01;
aff1Si[599, 0] := 9.95000E+03; aff1Si[599, 1] := 1.91898E-01;
aff1Si[600, 0] := 1.00000E+04; aff1Si[600, 1] := 1.90581E-01;
aff1Si[601, 0] := 1.00500E+04; aff1Si[601, 1] := 1.89274E-01;
aff1Si[602, 0] := 1.01000E+04; aff1Si[602, 1] := 1.87977E-01;
aff1Si[603, 0] := 1.01500E+04; aff1Si[603, 1] := 1.86690E-01;
aff1Si[604, 0] := 1.02000E+04; aff1Si[604, 1] := 1.85413E-01;
aff1Si[605, 0] := 1.02500E+04; aff1Si[605, 1] := 1.84146E-01;
aff1Si[606, 0] := 1.03000E+04; aff1Si[606, 1] := 1.82889E-01;
aff1Si[607, 0] := 1.03500E+04; aff1Si[607, 1] := 1.81642E-01;
aff1Si[608, 0] := 1.04000E+04; aff1Si[608, 1] := 1.80405E-01;
aff1Si[609, 0] := 1.04500E+04; aff1Si[609, 1] := 1.79177E-01;
aff1Si[610, 0] := 1.05000E+04; aff1Si[610, 1] := 1.77960E-01;
aff1Si[611, 0] := 1.05500E+04; aff1Si[611, 1] := 1.76752E-01;
aff1Si[612, 0] := 1.06000E+04; aff1Si[612, 1] := 1.75554E-01;
aff1Si[613, 0] := 1.06500E+04; aff1Si[613, 1] := 1.74366E-01;
aff1Si[614, 0] := 1.07000E+04; aff1Si[614, 1] := 1.73188E-01;
aff1Si[615, 0] := 1.07500E+04; aff1Si[615, 1] := 1.72019E-01;
aff1Si[616, 0] := 1.08000E+04; aff1Si[616, 1] := 1.70860E-01;
aff1Si[617, 0] := 1.08500E+04; aff1Si[617, 1] := 1.69710E-01;
aff1Si[618, 0] := 1.09000E+04; aff1Si[618, 1] := 1.68570E-01;
aff1Si[619, 0] := 1.09500E+04; aff1Si[619, 1] := 1.67439E-01;
aff1Si[620, 0] := 1.10000E+04; aff1Si[620, 1] := 1.66317E-01;
aff1Si[621, 0] := 1.10500E+04; aff1Si[621, 1] := 1.65205E-01;
aff1Si[622, 0] := 1.11000E+04; aff1Si[622, 1] := 1.64101E-01;
aff1Si[623, 0] := 1.11500E+04; aff1Si[623, 1] := 1.63007E-01;
aff1Si[624, 0] := 1.12000E+04; aff1Si[624, 1] := 1.61922E-01;
aff1Si[625, 0] := 1.12500E+04; aff1Si[625, 1] := 1.60846E-01;
aff1Si[626, 0] := 1.13000E+04; aff1Si[626, 1] := 1.59779E-01;
aff1Si[627, 0] := 1.13500E+04; aff1Si[627, 1] := 1.58721E-01;
aff1Si[628, 0] := 1.14000E+04; aff1Si[628, 1] := 1.57672E-01;
aff1Si[629, 0] := 1.14500E+04; aff1Si[629, 1] := 1.56631E-01;
aff1Si[630, 0] := 1.15000E+04; aff1Si[630, 1] := 1.55599E-01;
aff1Si[631, 0] := 1.15500E+04; aff1Si[631, 1] := 1.54575E-01;
aff1Si[632, 0] := 1.16000E+04; aff1Si[632, 1] := 1.53560E-01;
aff1Si[633, 0] := 1.16500E+04; aff1Si[633, 1] := 1.52553E-01;
aff1Si[634, 0] := 1.17000E+04; aff1Si[634, 1] := 1.51555E-01;
aff1Si[635, 0] := 1.17500E+04; aff1Si[635, 1] := 1.50565E-01;
aff1Si[636, 0] := 1.18000E+04; aff1Si[636, 1] := 1.49583E-01;
aff1Si[637, 0] := 1.18500E+04; aff1Si[637, 1] := 1.48610E-01;
aff1Si[638, 0] := 1.19000E+04; aff1Si[638, 1] := 1.47644E-01;
aff1Si[639, 0] := 1.19500E+04; aff1Si[639, 1] := 1.46686E-01;
aff1Si[640, 0] := 1.20000E+04; aff1Si[640, 1] := 1.45737E-01;
aff1Si[641, 0] := 1.20500E+04; aff1Si[641, 1] := 1.44795E-01;
aff1Si[642, 0] := 1.21000E+04; aff1Si[642, 1] := 1.43861E-01;
aff1Si[643, 0] := 1.21500E+04; aff1Si[643, 1] := 1.42934E-01;
aff1Si[644, 0] := 1.22000E+04; aff1Si[644, 1] := 1.42016E-01;
aff1Si[645, 0] := 1.22500E+04; aff1Si[645, 1] := 1.41104E-01;
aff1Si[646, 0] := 1.23000E+04; aff1Si[646, 1] := 1.40201E-01;
aff1Si[647, 0] := 1.23500E+04; aff1Si[647, 1] := 1.39305E-01;
aff1Si[648, 0] := 1.24000E+04; aff1Si[648, 1] := 1.38416E-01;
aff1Si[649, 0] := 1.24500E+04; aff1Si[649, 1] := 1.37534E-01;
aff1Si[650, 0] := 1.25000E+04; aff1Si[650, 1] := 1.36659E-01;
aff1Si[651, 0] := 1.25500E+04; aff1Si[651, 1] := 1.35792E-01;
aff1Si[652, 0] := 1.26000E+04; aff1Si[652, 1] := 1.34932E-01;
aff1Si[653, 0] := 1.26500E+04; aff1Si[653, 1] := 1.34079E-01;
aff1Si[654, 0] := 1.27000E+04; aff1Si[654, 1] := 1.33233E-01;
aff1Si[655, 0] := 1.27500E+04; aff1Si[655, 1] := 1.32393E-01;
aff1Si[656, 0] := 1.28000E+04; aff1Si[656, 1] := 1.31561E-01;
aff1Si[657, 0] := 1.28500E+04; aff1Si[657, 1] := 1.30735E-01;
aff1Si[658, 0] := 1.29000E+04; aff1Si[658, 1] := 1.29916E-01;
aff1Si[659, 0] := 1.29500E+04; aff1Si[659, 1] := 1.29103E-01;
aff1Si[660, 0] := 1.30000E+04; aff1Si[660, 1] := 1.28297E-01;
aff1Si[661, 0] := 1.30500E+04; aff1Si[661, 1] := 1.27498E-01;
aff1Si[662, 0] := 1.31000E+04; aff1Si[662, 1] := 1.26705E-01;
aff1Si[663, 0] := 1.31500E+04; aff1Si[663, 1] := 1.25918E-01;
aff1Si[664, 0] := 1.32000E+04; aff1Si[664, 1] := 1.25137E-01;
aff1Si[665, 0] := 1.32500E+04; aff1Si[665, 1] := 1.24363E-01;
aff1Si[666, 0] := 1.33000E+04; aff1Si[666, 1] := 1.23595E-01;
aff1Si[667, 0] := 1.33500E+04; aff1Si[667, 1] := 1.22833E-01;
aff1Si[668, 0] := 1.34000E+04; aff1Si[668, 1] := 1.22078E-01;
aff1Si[669, 0] := 1.34500E+04; aff1Si[669, 1] := 1.21328E-01;
aff1Si[670, 0] := 1.35000E+04; aff1Si[670, 1] := 1.20584E-01;
aff1Si[671, 0] := 1.35500E+04; aff1Si[671, 1] := 1.19846E-01;
aff1Si[672, 0] := 1.36000E+04; aff1Si[672, 1] := 1.19114E-01;
aff1Si[673, 0] := 1.36500E+04; aff1Si[673, 1] := 1.18387E-01;
aff1Si[674, 0] := 1.37000E+04; aff1Si[674, 1] := 1.17667E-01;
aff1Si[675, 0] := 1.37500E+04; aff1Si[675, 1] := 1.16952E-01;
aff1Si[676, 0] := 1.38000E+04; aff1Si[676, 1] := 1.16242E-01;
aff1Si[677, 0] := 1.38500E+04; aff1Si[677, 1] := 1.15538E-01;
aff1Si[678, 0] := 1.39000E+04; aff1Si[678, 1] := 1.14840E-01;
aff1Si[679, 0] := 1.39500E+04; aff1Si[679, 1] := 1.14147E-01;
aff1Si[680, 0] := 1.40000E+04; aff1Si[680, 1] := 1.13459E-01;
aff1Si[681, 0] := 1.40500E+04; aff1Si[681, 1] := 1.12777E-01;
aff1Si[682, 0] := 1.41000E+04; aff1Si[682, 1] := 1.12100E-01;
aff1Si[683, 0] := 1.41500E+04; aff1Si[683, 1] := 1.11428E-01;
aff1Si[684, 0] := 1.42000E+04; aff1Si[684, 1] := 1.10762E-01;
aff1Si[685, 0] := 1.42500E+04; aff1Si[685, 1] := 1.10101E-01;
aff1Si[686, 0] := 1.43000E+04; aff1Si[686, 1] := 1.09444E-01;
aff1Si[687, 0] := 1.43500E+04; aff1Si[687, 1] := 1.08793E-01;
aff1Si[688, 0] := 1.44000E+04; aff1Si[688, 1] := 1.08147E-01;
aff1Si[689, 0] := 1.44500E+04; aff1Si[689, 1] := 1.07505E-01;
aff1Si[690, 0] := 1.45000E+04; aff1Si[690, 1] := 1.06869E-01;
aff1Si[691, 0] := 1.45500E+04; aff1Si[691, 1] := 1.06237E-01;
aff1Si[692, 0] := 1.46000E+04; aff1Si[692, 1] := 1.05610E-01;
aff1Si[693, 0] := 1.46500E+04; aff1Si[693, 1] := 1.04988E-01;
aff1Si[694, 0] := 1.47000E+04; aff1Si[694, 1] := 1.04371E-01;
aff1Si[695, 0] := 1.47500E+04; aff1Si[695, 1] := 1.03758E-01;
aff1Si[696, 0] := 1.48000E+04; aff1Si[696, 1] := 1.03150E-01;
aff1Si[697, 0] := 1.48500E+04; aff1Si[697, 1] := 1.02546E-01;
aff1Si[698, 0] := 1.49000E+04; aff1Si[698, 1] := 1.01947E-01;
aff1Si[699, 0] := 1.49500E+04; aff1Si[699, 1] := 1.01352E-01;
aff1Si[700, 0] := 1.50000E+04; aff1Si[700, 1] := 1.00762E-01;
aff1Si[701, 0] := 1.50500E+04; aff1Si[701, 1] := 1.00177E-01;
aff1Si[702, 0] := 1.51000E+04; aff1Si[702, 1] := 9.95951E-02;
aff1Si[703, 0] := 1.51500E+04; aff1Si[703, 1] := 9.90180E-02;
aff1Si[704, 0] := 1.52000E+04; aff1Si[704, 1] := 9.84451E-02;
aff1Si[705, 0] := 1.52500E+04; aff1Si[705, 1] := 9.78765E-02;
aff1Si[706, 0] := 1.53000E+04; aff1Si[706, 1] := 9.73121E-02;
aff1Si[707, 0] := 1.53500E+04; aff1Si[707, 1] := 9.67518E-02;
aff1Si[708, 0] := 1.54000E+04; aff1Si[708, 1] := 9.61956E-02;
aff1Si[709, 0] := 1.54500E+04; aff1Si[709, 1] := 9.56435E-02;
aff1Si[710, 0] := 1.55000E+04; aff1Si[710, 1] := 9.50954E-02;
aff1Si[711, 0] := 1.55500E+04; aff1Si[711, 1] := 9.45513E-02;
aff1Si[712, 0] := 1.56000E+04; aff1Si[712, 1] := 9.40112E-02;
aff1Si[713, 0] := 1.56500E+04; aff1Si[713, 1] := 9.34750E-02;
aff1Si[714, 0] := 1.57000E+04; aff1Si[714, 1] := 9.29426E-02;
aff1Si[715, 0] := 1.57500E+04; aff1Si[715, 1] := 9.24142E-02;
aff1Si[716, 0] := 1.58000E+04; aff1Si[716, 1] := 9.18895E-02;
aff1Si[717, 0] := 1.58500E+04; aff1Si[717, 1] := 9.13686E-02;
aff1Si[718, 0] := 1.59000E+04; aff1Si[718, 1] := 9.08515E-02;
aff1Si[719, 0] := 1.59500E+04; aff1Si[719, 1] := 9.03380E-02;
aff1Si[720, 0] := 1.60000E+04; aff1Si[720, 1] := 8.98282E-02;
aff1Si[721, 0] := 1.60500E+04; aff1Si[721, 1] := 8.93220E-02;
aff1Si[722, 0] := 1.61000E+04; aff1Si[722, 1] := 8.88195E-02;
aff1Si[723, 0] := 1.61500E+04; aff1Si[723, 1] := 8.83205E-02;
aff1Si[724, 0] := 1.62000E+04; aff1Si[724, 1] := 8.78251E-02;
aff1Si[725, 0] := 1.62500E+04; aff1Si[725, 1] := 8.73331E-02;
aff1Si[726, 0] := 1.63000E+04; aff1Si[726, 1] := 8.68446E-02;
aff1Si[727, 0] := 1.63500E+04; aff1Si[727, 1] := 8.63595E-02;
aff1Si[728, 0] := 1.64000E+04; aff1Si[728, 1] := 8.58779E-02;
aff1Si[729, 0] := 1.64500E+04; aff1Si[729, 1] := 8.53996E-02;
aff1Si[730, 0] := 1.65000E+04; aff1Si[730, 1] := 8.49247E-02;
aff1Si[731, 0] := 1.65500E+04; aff1Si[731, 1] := 8.44530E-02;
aff1Si[732, 0] := 1.66000E+04; aff1Si[732, 1] := 8.39847E-02;
aff1Si[733, 0] := 1.66500E+04; aff1Si[733, 1] := 8.35196E-02;
aff1Si[734, 0] := 1.67000E+04; aff1Si[734, 1] := 8.30578E-02;
aff1Si[735, 0] := 1.67500E+04; aff1Si[735, 1] := 8.25991E-02;
aff1Si[736, 0] := 1.68000E+04; aff1Si[736, 1] := 8.21436E-02;
aff1Si[737, 0] := 1.68500E+04; aff1Si[737, 1] := 8.16913E-02;
aff1Si[738, 0] := 1.69000E+04; aff1Si[738, 1] := 8.12420E-02;
aff1Si[739, 0] := 1.69500E+04; aff1Si[739, 1] := 8.07959E-02;
aff1Si[740, 0] := 1.70000E+04; aff1Si[740, 1] := 8.03528E-02;
aff1Si[741, 0] := 1.70500E+04; aff1Si[741, 1] := 7.99127E-02;
aff1Si[742, 0] := 1.71000E+04; aff1Si[742, 1] := 7.94756E-02;
aff1Si[743, 0] := 1.71500E+04; aff1Si[743, 1] := 7.90415E-02;
aff1Si[744, 0] := 1.72000E+04; aff1Si[744, 1] := 7.86103E-02;
aff1Si[745, 0] := 1.72500E+04; aff1Si[745, 1] := 7.81820E-02;
aff1Si[746, 0] := 1.73000E+04; aff1Si[746, 1] := 7.77567E-02;
aff1Si[747, 0] := 1.73500E+04; aff1Si[747, 1] := 7.73342E-02;
aff1Si[748, 0] := 1.74000E+04; aff1Si[748, 1] := 7.69145E-02;
aff1Si[749, 0] := 1.74500E+04; aff1Si[749, 1] := 7.64977E-02;
aff1Si[750, 0] := 1.75000E+04; aff1Si[750, 1] := 7.60836E-02;
aff1Si[751, 0] := 1.75500E+04; aff1Si[751, 1] := 7.56724E-02;
aff1Si[752, 0] := 1.76000E+04; aff1Si[752, 1] := 7.52639E-02;
aff1Si[753, 0] := 1.76500E+04; aff1Si[753, 1] := 7.48580E-02;
aff1Si[754, 0] := 1.77000E+04; aff1Si[754, 1] := 7.44549E-02;
aff1Si[755, 0] := 1.77500E+04; aff1Si[755, 1] := 7.40544E-02;
aff1Si[756, 0] := 1.78000E+04; aff1Si[756, 1] := 7.36566E-02;
aff1Si[757, 0] := 1.78500E+04; aff1Si[757, 1] := 7.32614E-02;
aff1Si[758, 0] := 1.79000E+04; aff1Si[758, 1] := 7.28688E-02;
aff1Si[759, 0] := 1.79500E+04; aff1Si[759, 1] := 7.24788E-02;
aff1Si[760, 0] := 1.80000E+04; aff1Si[760, 1] := 7.20914E-02;
aff1Si[761, 0] := 1.80500E+04; aff1Si[761, 1] := 7.17065E-02;
aff1Si[762, 0] := 1.81000E+04; aff1Si[762, 1] := 7.13242E-02;
aff1Si[763, 0] := 1.81500E+04; aff1Si[763, 1] := 7.09443E-02;
aff1Si[764, 0] := 1.82000E+04; aff1Si[764, 1] := 7.05669E-02;
aff1Si[765, 0] := 1.82500E+04; aff1Si[765, 1] := 7.01919E-02;
aff1Si[766, 0] := 1.83000E+04; aff1Si[766, 1] := 6.98193E-02;
aff1Si[767, 0] := 1.83500E+04; aff1Si[767, 1] := 6.94492E-02;
aff1Si[768, 0] := 1.84000E+04; aff1Si[768, 1] := 6.90814E-02;
aff1Si[769, 0] := 1.84500E+04; aff1Si[769, 1] := 6.87160E-02;
aff1Si[770, 0] := 1.85000E+04; aff1Si[770, 1] := 6.83530E-02;
aff1Si[771, 0] := 1.85500E+04; aff1Si[771, 1] := 6.79922E-02;
aff1Si[772, 0] := 1.86000E+04; aff1Si[772, 1] := 6.76338E-02;
aff1Si[773, 0] := 1.86500E+04; aff1Si[773, 1] := 6.72777E-02;
aff1Si[774, 0] := 1.87000E+04; aff1Si[774, 1] := 6.69238E-02;
aff1Si[775, 0] := 1.87500E+04; aff1Si[775, 1] := 6.65723E-02;
aff1Si[776, 0] := 1.88000E+04; aff1Si[776, 1] := 6.62229E-02;
aff1Si[777, 0] := 1.88500E+04; aff1Si[777, 1] := 6.58758E-02;
aff1Si[778, 0] := 1.89000E+04; aff1Si[778, 1] := 6.55308E-02;
aff1Si[779, 0] := 1.89500E+04; aff1Si[779, 1] := 6.51880E-02;
aff1Si[780, 0] := 1.90000E+04; aff1Si[780, 1] := 6.48474E-02;
aff1Si[781, 0] := 1.90500E+04; aff1Si[781, 1] := 6.45089E-02;
aff1Si[782, 0] := 1.91000E+04; aff1Si[782, 1] := 6.41725E-02;
aff1Si[783, 0] := 1.91500E+04; aff1Si[783, 1] := 6.38382E-02;
aff1Si[784, 0] := 1.92000E+04; aff1Si[784, 1] := 6.35060E-02;
aff1Si[785, 0] := 1.92500E+04; aff1Si[785, 1] := 6.31759E-02;
aff1Si[786, 0] := 1.93000E+04; aff1Si[786, 1] := 6.28478E-02;
aff1Si[787, 0] := 1.93500E+04; aff1Si[787, 1] := 6.25218E-02;
aff1Si[788, 0] := 1.94000E+04; aff1Si[788, 1] := 6.21978E-02;
aff1Si[789, 0] := 1.94500E+04; aff1Si[789, 1] := 6.18758E-02;
aff1Si[790, 0] := 1.95000E+04; aff1Si[790, 1] := 6.15557E-02;
aff1Si[791, 0] := 1.95500E+04; aff1Si[791, 1] := 6.12377E-02;
aff1Si[792, 0] := 1.96000E+04; aff1Si[792, 1] := 6.09216E-02;
aff1Si[793, 0] := 1.96500E+04; aff1Si[793, 1] := 6.06075E-02;
aff1Si[794, 0] := 1.97000E+04; aff1Si[794, 1] := 6.02953E-02;
aff1Si[795, 0] := 1.97500E+04; aff1Si[795, 1] := 5.99849E-02;
aff1Si[796, 0] := 1.98000E+04; aff1Si[796, 1] := 5.96765E-02;
aff1Si[797, 0] := 1.98500E+04; aff1Si[797, 1] := 5.93699E-02;
aff1Si[798, 0] := 1.99000E+04; aff1Si[798, 1] := 5.90652E-02;
aff1Si[799, 0] := 1.99500E+04; aff1Si[799, 1] := 5.87623E-02;
aff1Si[800, 0] := 2.00000E+04; aff1Si[800, 1] := 5.84613E-02;
aff1Si[801, 0] := 2.00500E+04; aff1Si[801, 1] := 5.81622E-02;
aff1Si[802, 0] := 2.01000E+04; aff1Si[802, 1] := 5.78648E-02;
aff1Si[803, 0] := 2.01500E+04; aff1Si[803, 1] := 5.75692E-02;
aff1Si[804, 0] := 2.02000E+04; aff1Si[804, 1] := 5.72754E-02;
aff1Si[805, 0] := 2.02500E+04; aff1Si[805, 1] := 5.69833E-02;
aff1Si[806, 0] := 2.03000E+04; aff1Si[806, 1] := 5.66930E-02;
aff1Si[807, 0] := 2.03500E+04; aff1Si[807, 1] := 5.64044E-02;
aff1Si[808, 0] := 2.04000E+04; aff1Si[808, 1] := 5.61175E-02;
aff1Si[809, 0] := 2.04500E+04; aff1Si[809, 1] := 5.58323E-02;
aff1Si[810, 0] := 2.05000E+04; aff1Si[810, 1] := 5.55488E-02;
aff1Si[811, 0] := 2.05500E+04; aff1Si[811, 1] := 5.52670E-02;
aff1Si[812, 0] := 2.06000E+04; aff1Si[812, 1] := 5.49869E-02;
aff1Si[813, 0] := 2.06500E+04; aff1Si[813, 1] := 5.47084E-02;
aff1Si[814, 0] := 2.07000E+04; aff1Si[814, 1] := 5.44316E-02;
aff1Si[815, 0] := 2.07500E+04; aff1Si[815, 1] := 5.41564E-02;
aff1Si[816, 0] := 2.08000E+04; aff1Si[816, 1] := 5.38828E-02;
aff1Si[817, 0] := 2.08500E+04; aff1Si[817, 1] := 5.36108E-02;
aff1Si[818, 0] := 2.09000E+04; aff1Si[818, 1] := 5.33404E-02;
aff1Si[819, 0] := 2.09500E+04; aff1Si[819, 1] := 5.30716E-02;
aff1Si[820, 0] := 2.10000E+04; aff1Si[820, 1] := 5.28044E-02;
aff1Si[821, 0] := 2.10500E+04; aff1Si[821, 1] := 5.25387E-02;
aff1Si[822, 0] := 2.11000E+04; aff1Si[822, 1] := 5.22745E-02;
aff1Si[823, 0] := 2.11500E+04; aff1Si[823, 1] := 5.20119E-02;
aff1Si[824, 0] := 2.12000E+04; aff1Si[824, 1] := 5.17508E-02;
aff1Si[825, 0] := 2.12500E+04; aff1Si[825, 1] := 5.14912E-02;
aff1Si[826, 0] := 2.13000E+04; aff1Si[826, 1] := 5.12332E-02;
aff1Si[827, 0] := 2.13500E+04; aff1Si[827, 1] := 5.09765E-02;
aff1Si[828, 0] := 2.14000E+04; aff1Si[828, 1] := 5.07214E-02;
aff1Si[829, 0] := 2.14500E+04; aff1Si[829, 1] := 5.04677E-02;
aff1Si[830, 0] := 2.15000E+04; aff1Si[830, 1] := 5.02155E-02;
aff1Si[831, 0] := 2.15500E+04; aff1Si[831, 1] := 4.99648E-02;
aff1Si[832, 0] := 2.16000E+04; aff1Si[832, 1] := 4.97154E-02;
aff1Si[833, 0] := 2.16500E+04; aff1Si[833, 1] := 4.94675E-02;
aff1Si[834, 0] := 2.17000E+04; aff1Si[834, 1] := 4.92210E-02;
aff1Si[835, 0] := 2.17500E+04; aff1Si[835, 1] := 4.89760E-02;
aff1Si[836, 0] := 2.18000E+04; aff1Si[836, 1] := 4.87323E-02;
aff1Si[837, 0] := 2.18500E+04; aff1Si[837, 1] := 4.84899E-02;
aff1Si[838, 0] := 2.19000E+04; aff1Si[838, 1] := 4.82490E-02;
aff1Si[839, 0] := 2.19500E+04; aff1Si[839, 1] := 4.80094E-02;
aff1Si[840, 0] := 2.20000E+04; aff1Si[840, 1] := 4.77712E-02;
aff1Si[841, 0] := 2.20500E+04; aff1Si[841, 1] := 4.75343E-02;
aff1Si[842, 0] := 2.21000E+04; aff1Si[842, 1] := 4.72987E-02;
aff1Si[843, 0] := 2.21500E+04; aff1Si[843, 1] := 4.70645E-02;
aff1Si[844, 0] := 2.22000E+04; aff1Si[844, 1] := 4.68315E-02;
aff1Si[845, 0] := 2.22500E+04; aff1Si[845, 1] := 4.65999E-02;
aff1Si[846, 0] := 2.23000E+04; aff1Si[846, 1] := 4.63696E-02;
aff1Si[847, 0] := 2.23500E+04; aff1Si[847, 1] := 4.61406E-02;
aff1Si[848, 0] := 2.24000E+04; aff1Si[848, 1] := 4.59128E-02;
aff1Si[849, 0] := 2.24500E+04; aff1Si[849, 1] := 4.56863E-02;
aff1Si[850, 0] := 2.25000E+04; aff1Si[850, 1] := 4.54611E-02;
aff1Si[851, 0] := 2.25500E+04; aff1Si[851, 1] := 4.52371E-02;
aff1Si[852, 0] := 2.26000E+04; aff1Si[852, 1] := 4.50144E-02;
aff1Si[853, 0] := 2.26500E+04; aff1Si[853, 1] := 4.47929E-02;
aff1Si[854, 0] := 2.27000E+04; aff1Si[854, 1] := 4.45726E-02;
aff1Si[855, 0] := 2.27500E+04; aff1Si[855, 1] := 4.43536E-02;
aff1Si[856, 0] := 2.28000E+04; aff1Si[856, 1] := 4.41357E-02;
aff1Si[857, 0] := 2.28500E+04; aff1Si[857, 1] := 4.39191E-02;
aff1Si[858, 0] := 2.29000E+04; aff1Si[858, 1] := 4.37037E-02;
aff1Si[859, 0] := 2.29500E+04; aff1Si[859, 1] := 4.34894E-02;
aff1Si[860, 0] := 2.30000E+04; aff1Si[860, 1] := 4.32763E-02;
aff1Si[861, 0] := 2.30500E+04; aff1Si[861, 1] := 4.30644E-02;
aff1Si[862, 0] := 2.31000E+04; aff1Si[862, 1] := 4.28537E-02;
aff1Si[863, 0] := 2.31500E+04; aff1Si[863, 1] := 4.26441E-02;
aff1Si[864, 0] := 2.32000E+04; aff1Si[864, 1] := 4.24357E-02;
aff1Si[865, 0] := 2.32500E+04; aff1Si[865, 1] := 4.22284E-02;
aff1Si[866, 0] := 2.33000E+04; aff1Si[866, 1] := 4.20222E-02;
aff1Si[867, 0] := 2.33500E+04; aff1Si[867, 1] := 4.18172E-02;
aff1Si[868, 0] := 2.34000E+04; aff1Si[868, 1] := 4.16133E-02;
aff1Si[869, 0] := 2.34500E+04; aff1Si[869, 1] := 4.14105E-02;
aff1Si[870, 0] := 2.35000E+04; aff1Si[870, 1] := 4.12089E-02;
aff1Si[871, 0] := 2.35500E+04; aff1Si[871, 1] := 4.10083E-02;
aff1Si[872, 0] := 2.36000E+04; aff1Si[872, 1] := 4.08089E-02;
aff1Si[873, 0] := 2.36500E+04; aff1Si[873, 1] := 4.06105E-02;
aff1Si[874, 0] := 2.37000E+04; aff1Si[874, 1] := 4.04132E-02;
aff1Si[875, 0] := 2.37500E+04; aff1Si[875, 1] := 4.02170E-02;
aff1Si[876, 0] := 2.38000E+04; aff1Si[876, 1] := 4.00218E-02;
aff1Si[877, 0] := 2.38500E+04; aff1Si[877, 1] := 3.98278E-02;
aff1Si[878, 0] := 2.39000E+04; aff1Si[878, 1] := 3.96347E-02;
aff1Si[879, 0] := 2.39500E+04; aff1Si[879, 1] := 3.94428E-02;
aff1Si[880, 0] := 2.40000E+04; aff1Si[880, 1] := 3.92519E-02;
aff1Si[881, 0] := 2.40500E+04; aff1Si[881, 1] := 3.90620E-02;
aff1Si[882, 0] := 2.41000E+04; aff1Si[882, 1] := 3.88732E-02;
aff1Si[883, 0] := 2.41500E+04; aff1Si[883, 1] := 3.86855E-02;
aff1Si[884, 0] := 2.42000E+04; aff1Si[884, 1] := 3.84988E-02;
aff1Si[885, 0] := 2.42500E+04; aff1Si[885, 1] := 3.83131E-02;
aff1Si[886, 0] := 2.43000E+04; aff1Si[886, 1] := 3.81284E-02;
aff1Si[887, 0] := 2.43500E+04; aff1Si[887, 1] := 3.79448E-02;
aff1Si[888, 0] := 2.44000E+04; aff1Si[888, 1] := 3.77621E-02;
aff1Si[889, 0] := 2.44500E+04; aff1Si[889, 1] := 3.75805E-02;
aff1Si[890, 0] := 2.45000E+04; aff1Si[890, 1] := 3.73999E-02;
aff1Si[891, 0] := 2.45500E+04; aff1Si[891, 1] := 3.72204E-02;
aff1Si[892, 0] := 2.46000E+04; aff1Si[892, 1] := 3.70418E-02;
aff1Si[893, 0] := 2.46500E+04; aff1Si[893, 1] := 3.68643E-02;
aff1Si[894, 0] := 2.47000E+04; aff1Si[894, 1] := 3.66877E-02;
aff1Si[895, 0] := 2.47500E+04; aff1Si[895, 1] := 3.65122E-02;
aff1Si[896, 0] := 2.48000E+04; aff1Si[896, 1] := 3.63377E-02;
aff1Si[897, 0] := 2.48500E+04; aff1Si[897, 1] := 3.61642E-02;
aff1Si[898, 0] := 2.49000E+04; aff1Si[898, 1] := 3.59917E-02;
aff1Si[899, 0] := 2.49500E+04; aff1Si[899, 1] := 3.58202E-02;
aff1Si[900, 0] := 2.50000E+04; aff1Si[900, 1] := 3.56497E-02;
aff1Si[901, 0] := 2.50500E+04; aff1Si[901, 1] := 3.54802E-02;
aff1Si[902, 0] := 2.51000E+04; aff1Si[902, 1] := 3.53118E-02;
aff1Si[903, 0] := 2.51500E+04; aff1Si[903, 1] := 3.51443E-02;
aff1Si[904, 0] := 2.52000E+04; aff1Si[904, 1] := 3.49780E-02;
aff1Si[905, 0] := 2.52500E+04; aff1Si[905, 1] := 3.48126E-02;
aff1Si[906, 0] := 2.53000E+04; aff1Si[906, 1] := 3.46483E-02;
aff1Si[907, 0] := 2.53500E+04; aff1Si[907, 1] := 3.44851E-02;
aff1Si[908, 0] := 2.54000E+04; aff1Si[908, 1] := 3.43229E-02;
aff1Si[909, 0] := 2.54500E+04; aff1Si[909, 1] := 3.41618E-02;
aff1Si[910, 0] := 2.55000E+04; aff1Si[910, 1] := 3.40017E-02;
aff1Si[911, 0] := 2.55500E+04; aff1Si[911, 1] := 3.38428E-02;
aff1Si[912, 0] := 2.56000E+04; aff1Si[912, 1] := 3.36850E-02;
aff1Si[913, 0] := 2.56500E+04; aff1Si[913, 1] := 3.35284E-02;
aff1Si[914, 0] := 2.57000E+04; aff1Si[914, 1] := 3.33729E-02;
aff1Si[915, 0] := 2.57500E+04; aff1Si[915, 1] := 3.32187E-02;
aff1Si[916, 0] := 2.58000E+04; aff1Si[916, 1] := 3.30656E-02;
aff1Si[917, 0] := 2.58500E+04; aff1Si[917, 1] := 3.29139E-02;
aff1Si[918, 0] := 2.59000E+04; aff1Si[918, 1] := 3.27635E-02;
aff1Si[919, 0] := 2.59500E+04; aff1Si[919, 1] := 3.26145E-02;
aff1Si[920, 0] := 2.60000E+04; aff1Si[920, 1] := 3.24668E-02;
aff1Si[921, 0] := 2.60500E+04; aff1Si[921, 1] := 3.23207E-02;
aff1Si[922, 0] := 2.61000E+04; aff1Si[922, 1] := 3.21759E-02;
aff1Si[923, 0] := 2.61500E+04; aff1Si[923, 1] := 3.20321E-02;
aff1Si[924, 0] := 2.62000E+04; aff1Si[924, 1] := 3.18901E-02;
aff1Si[925, 0] := 2.62500E+04; aff1Si[925, 1] := 3.17506E-02;
aff1Si[926, 0] := 2.63000E+04; aff1Si[926, 1] := 3.16141E-02;
aff1Si[927, 0] := 2.63500E+04; aff1Si[927, 1] := 3.14812E-02;
aff1Si[928, 0] := 2.64000E+04; aff1Si[928, 1] := 3.13530E-02;
aff1Si[929, 0] := 2.64500E+04; aff1Si[929, 1] := 3.12278E-02;
aff1Si[930, 0] := 2.65000E+04; aff1Si[930, 1] := 3.11041E-02;
aff1Si[931, 0] := 2.65500E+04; aff1Si[931, 1] := 3.09802E-02;
aff1Si[932, 0] := 2.66000E+04; aff1Si[932, 1] := 3.08547E-02;
aff1Si[933, 0] := 2.66500E+04; aff1Si[933, 1] := 3.07262E-02;
aff1Si[934, 0] := 2.67000E+04; aff1Si[934, 1] := 3.05943E-02;
aff1Si[935, 0] := 2.67500E+04; aff1Si[935, 1] := 3.04595E-02;
aff1Si[936, 0] := 2.68000E+04; aff1Si[936, 1] := 3.03219E-02;
aff1Si[937, 0] := 2.68500E+04; aff1Si[937, 1] := 3.01819E-02;
aff1Si[938, 0] := 2.69000E+04; aff1Si[938, 1] := 3.00397E-02;
aff1Si[939, 0] := 2.69500E+04; aff1Si[939, 1] := 2.98955E-02;
aff1Si[940, 0] := 2.70000E+04; aff1Si[940, 1] := 2.97500E-02;
aff1Si[941, 0] := 2.70500E+04; aff1Si[941, 1] := 2.96038E-02;
aff1Si[942, 0] := 2.71000E+04; aff1Si[942, 1] := 2.94577E-02;
aff1Si[943, 0] := 2.71500E+04; aff1Si[943, 1] := 2.93123E-02;
aff1Si[944, 0] := 2.72000E+04; aff1Si[944, 1] := 2.91682E-02;
aff1Si[945, 0] := 2.72500E+04; aff1Si[945, 1] := 2.90254E-02;
aff1Si[946, 0] := 2.73000E+04; aff1Si[946, 1] := 2.88837E-02;
aff1Si[947, 0] := 2.73500E+04; aff1Si[947, 1] := 2.87429E-02;
aff1Si[948, 0] := 2.74000E+04; aff1Si[948, 1] := 2.86028E-02;
aff1Si[949, 0] := 2.74500E+04; aff1Si[949, 1] := 2.84630E-02;
aff1Si[950, 0] := 2.75000E+04; aff1Si[950, 1] := 2.83237E-02;
aff1Si[951, 0] := 2.75500E+04; aff1Si[951, 1] := 2.81849E-02;
aff1Si[952, 0] := 2.76000E+04; aff1Si[952, 1] := 2.80467E-02;
aff1Si[953, 0] := 2.76500E+04; aff1Si[953, 1] := 2.79090E-02;
aff1Si[954, 0] := 2.77000E+04; aff1Si[954, 1] := 2.77719E-02;
aff1Si[955, 0] := 2.77500E+04; aff1Si[955, 1] := 2.76356E-02;
aff1Si[956, 0] := 2.78000E+04; aff1Si[956, 1] := 2.74998E-02;
aff1Si[957, 0] := 2.78500E+04; aff1Si[957, 1] := 2.73647E-02;
aff1Si[958, 0] := 2.79000E+04; aff1Si[958, 1] := 2.72301E-02;
aff1Si[959, 0] := 2.79500E+04; aff1Si[959, 1] := 2.70961E-02;
aff1Si[960, 0] := 2.80000E+04; aff1Si[960, 1] := 2.69627E-02;
aff1Si[961, 0] := 2.80500E+04; aff1Si[961, 1] := 2.68299E-02;
aff1Si[962, 0] := 2.81000E+04; aff1Si[962, 1] := 2.66976E-02;
aff1Si[963, 0] := 2.81500E+04; aff1Si[963, 1] := 2.65660E-02;
aff1Si[964, 0] := 2.82000E+04; aff1Si[964, 1] := 2.64348E-02;
aff1Si[965, 0] := 2.82500E+04; aff1Si[965, 1] := 2.63043E-02;
aff1Si[966, 0] := 2.83000E+04; aff1Si[966, 1] := 2.61743E-02;
aff1Si[967, 0] := 2.83500E+04; aff1Si[967, 1] := 2.60449E-02;
aff1Si[968, 0] := 2.84000E+04; aff1Si[968, 1] := 2.59160E-02;
aff1Si[969, 0] := 2.84500E+04; aff1Si[969, 1] := 2.57877E-02;
aff1Si[970, 0] := 2.85000E+04; aff1Si[970, 1] := 2.56600E-02;
aff1Si[971, 0] := 2.85500E+04; aff1Si[971, 1] := 2.55328E-02;
aff1Si[972, 0] := 2.86000E+04; aff1Si[972, 1] := 2.54061E-02;
aff1Si[973, 0] := 2.86500E+04; aff1Si[973, 1] := 2.52800E-02;
aff1Si[974, 0] := 2.87000E+04; aff1Si[974, 1] := 2.51545E-02;
aff1Si[975, 0] := 2.87500E+04; aff1Si[975, 1] := 2.50295E-02;
aff1Si[976, 0] := 2.88000E+04; aff1Si[976, 1] := 2.49050E-02;
aff1Si[977, 0] := 2.88500E+04; aff1Si[977, 1] := 2.47810E-02;
aff1Si[978, 0] := 2.89000E+04; aff1Si[978, 1] := 2.46576E-02;
aff1Si[979, 0] := 2.89500E+04; aff1Si[979, 1] := 2.45347E-02;
aff1Si[980, 0] := 2.90000E+04; aff1Si[980, 1] := 2.44123E-02;
aff1Si[981, 0] := 2.90500E+04; aff1Si[981, 1] := 2.42904E-02;
aff1Si[982, 0] := 2.91000E+04; aff1Si[982, 1] := 2.41691E-02;
aff1Si[983, 0] := 2.91500E+04; aff1Si[983, 1] := 2.40483E-02;
aff1Si[984, 0] := 2.92000E+04; aff1Si[984, 1] := 2.39279E-02;
aff1Si[985, 0] := 2.92500E+04; aff1Si[985, 1] := 2.38081E-02;
aff1Si[986, 0] := 2.93000E+04; aff1Si[986, 1] := 2.36888E-02;
aff1Si[987, 0] := 2.93500E+04; aff1Si[987, 1] := 2.35700E-02;
aff1Si[988, 0] := 2.94000E+04; aff1Si[988, 1] := 2.34517E-02;
aff1Si[989, 0] := 2.94500E+04; aff1Si[989, 1] := 2.33339E-02;
aff1Si[990, 0] := 2.95000E+04; aff1Si[990, 1] := 2.32167E-02;
aff1Si[991, 0] := 2.95500E+04; aff1Si[991, 1] := 2.30998E-02;
aff1Si[992, 0] := 2.96000E+04; aff1Si[992, 1] := 2.29835E-02;
aff1Si[993, 0] := 2.96500E+04; aff1Si[993, 1] := 2.28677E-02;
aff1Si[994, 0] := 2.97000E+04; aff1Si[994, 1] := 2.27523E-02;
aff1Si[995, 0] := 2.97500E+04; aff1Si[995, 1] := 2.26375E-02;
aff1Si[996, 0] := 2.98000E+04; aff1Si[996, 1] := 2.25230E-02;
aff1Si[997, 0] := 2.98500E+04; aff1Si[997, 1] := 2.24091E-02;
aff1Si[998, 0] := 2.99000E+04; aff1Si[998, 1] := 2.22956E-02;
aff1Si[999, 0] := 2.99500E+04; aff1Si[999, 1] := 2.21826E-02;
END_METHOD


METHOD PRIVATE SetError
VAR_INPUT
    sMsg	: Tc2_System.T_MaxString;
END_VAR

bError := TRUE;
sErrorMsg := sMsg;
END_METHOD


PROPERTY Val : LREAL
GET

Val := ff1;
END_GET
END_PROPERTY

END_FUNCTION_BLOCK

(* stored: Version 1.1.0.1
   POU FB_f1Chantler: Id {912040aa-fdfa-4b0e-aefb-9fa7198a9d85}, SpecialFunc None
   Method ClearError: Id {3f73a964-2d47-48d0-89ae-96b322a187fc}
   Method FB_init: Id {30272d3e-4464-4bba-a035-9f10c800cbcf}
   Method GetEnergyAtIndex: Id {96323b97-ceb8-4488-ac08-b8eb8104faa3}
   Method GetError: Id {6705dbac-accd-4175-8568-5ab60567f1ef}
   Method GetErrorMsg: Id {0693506c-63d2-4b7b-912b-c58ccf786deb}
   Method Getf1AtIndex: Id {31cc284d-4c99-42bf-93c3-407c07773f7f}
   Method MakeTables: Id {0a710fc9-6b84-4699-a391-43f3331f588a}
   Method SetError: Id {f9b58c67-99ec-4e91-a689-437ed37bb956}
   Property Val: Id {a1b6dcbf-f0de-44ef-b8ff-5606431d00c1}
   Get Get: Id {564cca61-f236-4ad1-9473-9acbfc3a4256} *)
